// TwinCAT 3 PLC project P1
// ProgramVersion: 3.1.4024.0
// libraries:
//   Tc2_Standard, * (Beckhoff Automation GmbH)
//   Tc2_System, * (Beckhoff Automation GmbH)
//   Tc3_Module, * (Beckhoff Automation GmbH)
//   Tc3_PLCopen_OpcUa, * (Beckhoff Automation GmbH)
//   BeckhoffJsonReadWriter,1.0,fbarresi
// project tree:
//   Data_Types/ E_Errors2_ReactorSet.TcDUT, E_Errors_Module.TcDUT, E_Errors1_ReactorSet.TcDUT, E_Errors_Reactor.TcDUT, E_MachineState.TcDUT, E_PIDMode.TcDUT, E_ValveMode.TcDUT, ST_SeqResult_FAT.TcDUT, ST_Seq_FAT.TcDUT, ST_SeqSteps_FAT.TcDUT, ST_StepConfig_FAT.TcDUT, ST_StepSts_FAT.TcDUT
//   GVLs/ FAT.TcGVL, Global_Constants.TcGVL, Global_Variables.TcGVL, Set_Points_Interlocks.TcGVL
//   / PlcTask.TcTTO
//   POUs/ FB_Reactor.TcPOU, FB_Reactor_Set.TcPOU, FB_Reactor_Set_Ext_FAT.TcPOU, MAIN.TcPOU, P_Module.TcPOU
//   POUs/Functions/ F_AnalogIn.TcPOU, F_Concat3.TcPOU (not stored), F_Concat4.TcPOU (not stored), F_Error.TcPOU, F_Error_Check.TcPOU, F_Error_Range.TcPOU, F_IEConvert.TcPOU, F_LowestReal.TcPOU, F_HighestReal.TcPOU, F_Temperature.TcPOU
//   POUs/Function_Blocks/ FB_Door_Closed.TcPOU, FB_EdgeMonitor.TcPOU, FB_ReadWrite_Json.TcPOU, FB_ValveControl.TcPOU, FB_ValveStatus.TcPOU, FB_VFD.TcPOU, FB_Watchdog.TcPOU
// real-time tasks:
//   TASK PlcTask: cycle T#10ms, priority 20, ADS port 350
// I/O:
//   DEVICE Device 2 (EtherCAT Automation Protocol) (disabled), AmsNetId 10.0.2.15.2.1
//     Box 1 (Subscriber)
//     Box 2 (Publisher)
// variable links:
//   P1/P1 Instance <-> Device 2 (EtherCAT Automation Protocol)
//     PlcTask Inputs/P_Module.rs1.r1.fan_vfd_status <-> Inputs/DevState
//   P1/P1 Instance <-> Device 2 (EtherCAT Automation Protocol)/Box 1 (Subscriber)
//     PlcTask Inputs/P_Module.rs1.directive <-> RS1_Bytes/Inputs/VarData[0]
//     PlcTask Inputs/P_Module.rs1.rs_dead_air_pump_service_assigned <-> RS1_Bools/Inputs/VarData[1]
//     PlcTask Inputs/P_Module.rs1.rs_purge_assist_service_assigned <-> RS1_Bools/Inputs/VarData[3]
//     PlcTask Inputs/P_Module.rs1.rs_steam_system_service_assigned <-> RS1_Bools/Inputs/VarData[2]
//     PlcTask Inputs/P_Module.rs1.rs_vac_cooling_pump_service_assigned <-> RS1_Bools/Inputs/VarData[0]
//     PlcTask Inputs/P_Module.u_dead_air_pump_status <-> Module_Bytes/Inputs/VarData[1]
//     PlcTask Inputs/P_Module.u_module_generic_byte <-> Module_Bytes/Inputs/VarData[4]
//     PlcTask Inputs/P_Module.u_purge_assist_status <-> Module_Bytes/Inputs/VarData[3]
//     PlcTask Inputs/P_Module.u_steam_system_status <-> Module_Bytes/Inputs/VarData[2]
//     PlcTask Inputs/P_Module.u_vac_cooling_pump_status <-> Module_Bytes/Inputs/VarData[0]
//   P1/P1 Instance <-> Device 2 (EtherCAT Automation Protocol)/Box 2 (Publisher)
//     PlcTask Outputs/P_Module.rs1.r{1..4}.error_code <-> RS1_Dwords/Outputs/VarData[{1..4}]  (4 links)
//     PlcTask Outputs/P_Module.rs1.rs_adsorption <-> RS1_Bytes/Outputs/VarData[2]
//     PlcTask Outputs/P_Module.rs1.rs_air_repres <-> RS1_Bytes/Outputs/VarData[1]
//     PlcTask Outputs/P_Module.rs1.rs_dead_air_evac <-> RS1_Bytes/Outputs/VarData[3]
//     PlcTask Outputs/P_Module.rs1.rs_dead_air_pump_service_request <-> RS1_Bools/Outputs/VarData[1]
//     PlcTask Outputs/P_Module.rs1.rs_estop <-> RS1_Bytes/Outputs/VarData[6]
//     PlcTask Outputs/P_Module.rs1.rs_idle <-> RS1_Bytes/Outputs/VarData[0]
//     PlcTask Outputs/P_Module.rs1.rs_purge_assist_service_request <-> RS1_Bools/Outputs/VarData[3]
//     PlcTask Outputs/P_Module.rs1.rs_shutdown <-> RS1_Bytes/Outputs/VarData[7]
//     PlcTask Outputs/P_Module.rs1.rs_shutdown_evac <-> RS1_Bytes/Outputs/VarData[8]
//     PlcTask Outputs/P_Module.rs1.rs_steam_desorption <-> RS1_Bytes/Outputs/VarData[4]
//     PlcTask Outputs/P_Module.rs1.rs_steam_system_service_request <-> RS1_Bools/Outputs/VarData[2]
//     PlcTask Outputs/P_Module.rs1.rs_vac_cooling_pump_service_request <-> RS1_Bools/Outputs/VarData[0]
//     PlcTask Outputs/P_Module.rs1.rs_vacuum_cooling <-> RS1_Bytes/Outputs/VarData[5]

CONFIGURATION P1
    RESOURCE PLC ON TwinCAT3
        TASK PlcTask(INTERVAL := T#10ms, PRIORITY := 20);
        PROGRAM MAIN WITH PlcTask : MAIN;
    END_RESOURCE
END_CONFIGURATION

// ---- Data_Types/E_Errors2_ReactorSet.TcDUT
// P1 - E_Errors2_ReactorSet
// Rev 1.0 - October 31, 2024

TYPE E_Errors2_ReactorSet :
(
	errTBD								:= 0
);
END_TYPE

// ---- Data_Types/E_Errors_Module.TcDUT
// P1 - E_Errors_Module
// Rev 1.0 - October 15, 2024

TYPE E_Errors_Module :
(
	errInletCO2				         		:= 0,    
	errInletH2O,  
	errOutletH2O,			                 
	errSteamManifoldLinePres,    
	errFilterDiffPres,       
	errSorbentDiffPres,
	errReactorWallTemp,
	errInletAirTemp,
	errSteamTempNearRS1Temp,
	errSteamBypassValveNotInPos
);
END_TYPE

// ---- Data_Types/E_Errors1_ReactorSet.TcDUT
// P1 - E_Errors1_ReactorSet
// Rev 1.0 - October 31, 2024

TYPE E_Errors1_ReactorSet :
(
	errReactor								:= 0,			       
	errFanDiffPres,			       
	errOutletCO2,		         
	errReactorSetPres,		    
	errDoorsClosed,	       
	errRepresValvePosition,	 
	errDeadAirValvePosition,	 
	errPurgeValvePosition,	 
	errCoolingValvePosition,	 
	errSteamControlValvePosition,	 
	errSteamHeaderValvePosition,	 
	errDeadAirPumpServiceAssignmentLost,
	errPurgeAssistServiceAssignmentLost,
	errVacCoolingPumpServiceAssignmentLost,
	errSteamSystemServiceAssignmentLost,
	errAdsorptionFailedToCool,
	errEvacuationPresFailedToReachTarget,
	errReactorAboveMaxStoragePres,
	errReactorAboveMaxPres,
	errSorbentAboveMaxStorageTemp,
	errSorbentAboveMaxTemp,
	errInletTempAboveMaxAllowedTemp,	
	errInletTempBelowMinAllowedTemp,
	errInsufficientDesorptionVacuum,
	errInsufficientReactorPressure,
	errSteamRepressurizationOverPressure,
	errCoolingPressureTooHigh,
	errDeadAirValveSorbentTempTooHigh,
	errRepresValveSorbentTempTooHigh,
	errSteamHeaderValvePressureTooHigh,
	errRepresValveSteamValveOpen,
	errReactorLeak
);
END_TYPE

// ---- Data_Types/E_Errors_Reactor.TcDUT
// P1 - E_Errors_Reactor
// Rev 1.0 - October 15, 2024

TYPE E_Errors_Reactor :
(
	errInletDoorsClose						:= 0,
	errOutletDoorsClose,	
	errInletDoorsOpen,
	errOutletDoorsOpen,	
	errInletClampsRetract,	
	errOutletClampsRetract,
	errInletClampsExtend,
	errOutletClampsExtend,	
	errOutletLineTemp,
	errInletTopLeftTemp,		
	errInletTopRightTemp,	
	errInletBottomLeftTemp,	
	errInletBottomRightTemp,	
	errOutletTopLeftTemp,
	errOutletTopRightTemp,	
	errOutletBottomLeftTemp,	
	errOutletBottomRightTemp,
	errInletDoorsNotClosedForClamps,
	errOutletDoorsNotClosedForClamps,
	errInletClampsNotRetractedForDoors,
	errOutletClampsNotRetractedForDoors,
	errFanVFD,
	errFanRun
);
END_TYPE

// ---- Data_Types/E_MachineState.TcDUT
// P1 - E_MachineState
// Rev 1.0 - October 9, 2024

TYPE E_MachineState :
(
	eIdle						:= 0,
	eDeadAirEvacuation,
	eSteamDesorption,
	eVacuumCooling,
	eAirRepressurization,
	eAdsorption,
	eShutdown					:= 12,
	eShutdownEvac,
	eEmergencyStop
);
END_TYPE

// ---- Data_Types/E_PIDMode.TcDUT
// E_PIDMode
// Rev 1.0 - October 23, 2024

TYPE E_PIDMode :
(
	eOff						:= 0,
	eManual,
	eAuto,
	eTune
);
END_TYPE

// ---- Data_Types/E_ValveMode.TcDUT
// E_ValveMode
// Rev 1.0 - October 15, 2024

TYPE E_ValveMode :
(
	eClear						:= 0,
	eTransit,
	eError
);
END_TYPE

// ---- Data_Types/ST_SeqResult_FAT.TcDUT
TYPE ST_SeqResult_FAT :
STRUCT
	{attribute 'json' := 'TestName'}
	test_name : STRING;
	{attribute 'json' := 'TestDate'}
	test_date : STRING;
	{attribute 'json' := 'SeqSts'}
	status : STRING;
	{attribute 'json' := 'StepsCompleted'}
	steps : STRING;
	{attribute 'json' := 'error_id'}
	error : INT;
END_STRUCT
END_TYPE

// ---- Data_Types/ST_Seq_FAT.TcDUT
TYPE ST_Seq_FAT :
STRUCT
	{attribute 'json' := 'TestName'}
	test_name : STRING;
	{attribute 'json' := 'Step1'}
	step_1 : ST_SeqSteps_FAT;
	{attribute 'json' := 'Step2'}
	step_2 : ST_SeqSteps_FAT;
	{attribute 'json' := 'Step3'}
	step_3 : ST_SeqSteps_FAT;
	{attribute 'json' := 'Step4'}
	step_4 : ST_SeqSteps_FAT;
	{attribute 'json' := 'Step5'}
	step_5 : ST_SeqSteps_FAT;
	{attribute 'json' := 'Step6'}
	step_6 : ST_SeqSteps_FAT;
	{attribute 'json' := 'Step7'}
	step_7 : ST_SeqSteps_FAT;
	{attribute 'json' := 'Step8'}
	step_8 : ST_SeqSteps_FAT;
	{attribute 'json' := 'Step9'}
	step_9 : ST_SeqSteps_FAT;
	{attribute 'json' := 'Step10'}
	step_10 : ST_SeqSteps_FAT;
	
	
	
END_STRUCT
END_TYPE

// ---- Data_Types/ST_SeqSteps_FAT.TcDUT
TYPE ST_SeqSteps_FAT :
STRUCT
	{attribute 'json' := 'Summary'}
	summary : STRING(255);
	{attribute 'json' := 'Config'}
	config : ST_StepConfig_FAT;
END_STRUCT
END_TYPE

// ---- Data_Types/ST_StepConfig_FAT.TcDUT
TYPE ST_StepConfig_FAT :
STRUCT
	{attribute 'json' := 'react_pres'}
	react_press : REAL;
	{attribute 'json' := 'sorbent_temp'}
	sorbent_temp : REAL;
	{attribute 'json' := 'SP_1'}
	sp_1 : REAL;
	{attribute 'json' := 'SP_2'}
	sp_2 : REAL;
	{attribute 'json' := 'SP_3'}
	sp_3 : REAL;
	{attribute 'json' := 'SP_4'}
	sp_4 : REAL;
	{attribute 'json' := 'V_1'}
	valve_1 : STRING;
	{attribute 'json' := 'V_2'}
	valve_2 : STRING;
	{attribute 'json' := 'V_3'}
	valve_3 : STRING;
	{attribute 'json' := 'V_4'}
	valve_4 : STRING;
	{attribute 'json' := 'C_1'}
	check_1 : STRING;
	{attribute 'json' := 'C_2'}
	check_2 : STRING;
	{attribute 'json' := 'C_3'}
	check_3 : STRING;
	{attribute 'json' := 'C_4'}
	check_4 : STRING;
END_STRUCT
END_TYPE

// ---- Data_Types/ST_StepSts_FAT.TcDUT
TYPE ST_StepSts_FAT :
STRUCT
	{attribute 'json' := 'step_number'}
	step_number : INT;
	{attribute 'json' := 'react_pres'}
	react_press : REAL;
	{attribute 'json' := 'sorbent_temp'}
	sorbent_temp : REAL;
	{attribute 'json' := 'seq_sts'}
	seq_sts : STRING;
	
END_STRUCT
END_TYPE

// ---- GVLs/FAT.TcGVL
{attribute 'qualified_only'}
VAR_GLOBAL
	st_steam_desorption : ST_Seq_FAT;  // structure that parses the json file
	st_steam_desorption_result : ST_SeqResult_FAT;
	json_file_path : STRING(255) := 'C:/Users/asita/Documents/Steam_Desorption_FAT_Nominal.json';
END_VAR

// ---- GVLs/Global_Constants.TcGVL
// P1 - Global_Constants
// Rev 1.0 - November 2, 2024

VAR_GLOBAL CONSTANT
	
	_IDLE																: BYTE		:= 0;
	_STARTED															: BYTE		:= 1;
	_COMPLETED															: BYTE		:= 2;
	_ERROR																: BYTE		:= 9;
	
	_OPEN																: INT 		:= 100;
	_CLOSE																: INT		:= 0;
	
	_TEMP_VALID_TIME													: INT		:= 30;
	_VALVE_CHECK_TIME													: INT		:= 3000;

	_SECONDS															: REAL		:= 1000;
	_MINUTES															: REAL		:= 60000;
	
	_PERCENT_FACTOR														: REAL		:= 327.67;		// Factor to convert input to output percentage
	_VALVE_CLOSED														: INT		:= 3;
	_VALVE_OPEN															: INT		:= 95;

	_FAN_SPEED_MAX														: REAL		:= 1765;		// Maximum Fan RPM
	_FAN_SPEED_MIN														: REAL		:= 300;			// Minimum Fan RPM
	_FAN_ON																: REAL		:= 100;
	_FAN_START_TIME														: TIME		:= T#10S; 
	
	_DOOR_LATCH_CLOSE_TIME												: TIME		:= T#2S;

	_FAN_DELAY_TIME														: INT		:= 2000;
	_STOPPING_TIME														: REAL		:= 2000;

(*
	_DRAIN_TIME															: TIME		:= T#3S;
	_PUMP_SPEED_MAX														: REAL		:= 3540;		// Maximum Pump RPM
	_PUMP_SPEED_MIN														: REAL		:= 200;			// Minimum Pump RPM
	_FAN_RS_DELAY_TIME													: INT		:= 10000;
	_PAUSE_TIME															: REAL		:= 2000;
	_VALVE_TIME															: REAL		:= 3000;
	_FAN_SHUTDOWN_TIME													: REAL		:= 10000;
	_VALVE_INCREMENT_TIME												: REAL		:= 250;			// Time period for incremental change in valve position (mSecs)
	_VALVE_CLOSED														: INT		:= 3;
	_VALVE_OPEN															: INT		:= 95;
*)	
	_CURRENT_480_FACTOR													: REAL		:= 218.44;      // = 32767 counts / 150 amps
	_VOLTAGE_480_FACTOR													: REAL		:= 65.53;		// 0 - 500 VAC 
	_FAN_RPM_FACTOR														: REAL		:= 17.65;		// Factor to convert fan percent input to rpm output (max rpm / 100)

END_VAR

// ---- GVLs/Global_Variables.TcGVL
// P1 - Global_Variables
// Rev 1.0 - October 23, 2024

VAR_GLOBAL
	grDoorDelay															: REAL;
	grValveDelay														: REAL;
	grSteamControlValveDelay											: REAL;
	grClampDelay														: REAL;
	
	gbReset																: BOOL;
END_VAR

// ---- GVLs/Set_Points_Interlocks.TcGVL
// P1 - Set_Points_Interlocks
// Rev 1.0 - October 31, 2024

VAR_GLOBAL PERSISTENT
	
	{attribute 'OPC.UA.DA' := '1'}
	{attribute 'OPC.UA.DA.Access' := '1'}  				                
	IL_repres_valve_steam_valve_or										: BOOL;
	
	{attribute 'OPC.UA.DA' := '1'}
	SP_acceptable_reactor_pressure										: REAL;
	{attribute 'OPC.UA.DA' := '1'}
	SP_cooling_acceptable_pressure										: REAL;	
	{attribute 'OPC.UA.DA' := '1'}
	SP_cooling_target_pressure											: REAL;	
	{attribute 'OPC.UA.DA' := '1'}
	SP_clamp_extend_retract_duration									: REAL		:= 6;	
	{attribute 'OPC.UA.DA' := '1'}
	SP_door_open_close_duration											: REAL		:= 30;
	{attribute 'OPC.UA.DA' := '1'}
	SP_door_close_retries_before_error									: INT		:= 3;
	{attribute 'OPC.UA.DA' := '1'}
	SP_door_close_reset_duration										: REAL		:= 5;
	{attribute 'OPC.UA.DA' := '1'}	
	SP_evacuation_leak_test_acceptable_leak								: REAL		:= 0.2;
	{attribute 'OPC.UA.DA' := '1'}	
	SP_evacuation_leak_test_active										: BOOL;
	{attribute 'OPC.UA.DA' := '1'}	
	SP_evacuation_leak_test_duration									: REAL		:= 60;
	{attribute 'OPC.UA.DA' := '1'}
	SP_evacuation_target_pressure										: REAL;
	{attribute 'OPC.UA.DA' := '1'}
	SP_maximum_cooling_duration											: REAL;			
	{attribute 'OPC.UA.DA' := '1'}
	SP_maximum_desorption_sorbent_temperature							: REAL;			
	{attribute 'OPC.UA.DA' := '1'}	
	SP_maximum_evac_storage_pressure									: REAL;
	{attribute 'OPC.UA.DA' := '1'}	
	SP_maximum_evac_storage_temperature									: REAL;
	{attribute 'OPC.UA.DA' := '1'}
	SP_maximum_evacuation_duration										: REAL;
	{attribute 'OPC.UA.DA' := '1'}
	SP_maximum_inlet_air_temperature_during_adsorption					: REAL;						
	{attribute 'OPC.UA.DA' := '1'}
	SP_maximum_inlet_air_temperature									: REAL;
	{attribute 'OPC.UA.DA' := '1'}
	SP_maximum_pressure_for_steam_introduction							: REAL;
	{attribute 'OPC.UA.DA' := '1'}
	IL_maximum_pressure_for_steam_introduction_or						: BOOL;
	{attribute 'OPC.UA.DA' := '1'}
	{attribute 'OPC.UA.DA.Access' := '1'}  				                
	IL_maximum_pressure_for_steam_introduction_or_status				: BOOL;
	{attribute 'OPC.UA.DA' := '1'}
	SP_maximum_reactor_pressure											: REAL		:= 1.07;
	{attribute 'OPC.UA.DA' := '1'}
	IL_maximum_reactor_pressure_or										: BOOL;
	{attribute 'OPC.UA.DA' := '1'}
	{attribute 'OPC.UA.DA.Access' := '1'}  				                
	IL_maximum_reactor_pressure_or_status								: BOOL;
	{attribute 'OPC.UA.DA' := '1'}
	SP_maximum_reasonable_sorbent_TC_reading							: REAL;
	{attribute 'OPC.UA.DA' := '1'}
	SP_maximum_sorbent_temperature										: REAL;
	{attribute 'OPC.UA.DA' := '1'}
	IL_maximum_sorbent_temperature_or									: BOOL;
	{attribute 'OPC.UA.DA' := '1'}
	{attribute 'OPC.UA.DA.Access' := '1'}  				                
	IL_maximum_sorbent_temperature_or_status							: BOOL;
	{attribute 'OPC.UA.DA' := '1'}
	SP_maximum_sorbent_temperature_for_dead_air_line					: REAL;
	{attribute 'OPC.UA.DA' := '1'}
	IL_maximum_sorbent_temperature_for_dead_air_line_or					: BOOL;
	{attribute 'OPC.UA.DA' := '1'}
	{attribute 'OPC.UA.DA.Access' := '1'}  				                
	IL_maximum_sorbent_temperature_for_dead_air_line_or_status			: BOOL;
	{attribute 'OPC.UA.DA' := '1'}
	SP_maximum_sorbent_temperature_for_repressurization					: REAL;
	{attribute 'OPC.UA.DA' := '1'}
	IL_maximum_sorbent_temperature_for_repressurization_or				: BOOL;
	{attribute 'OPC.UA.DA' := '1'}
	{attribute 'OPC.UA.DA.Access' := '1'}  				                
	IL_maximum_sorbent_temperature_for_repressurization_or_status		: BOOL;
	{attribute 'OPC.UA.DA' := '1'}
	SP_maximum_steam_repressurization_duration							: REAL;
	{attribute 'OPC.UA.DA' := '1'}
	SP_minimum_evacuation_duration										: REAL;
	{attribute 'OPC.UA.DA' := '1'}
	SP_minimum_inlet_air_temperature									: REAL;
	{attribute 'OPC.UA.DA' := '1'}
	SP_minimum_reasonable_sorbent_TC_reading							: REAL;
	{attribute 'OPC.UA.DA' := '1'}
	SP_purge_duration													: REAL;
	{attribute 'OPC.UA.DA' := '1'}
	SP_steam_control_valve_open_close_duration							: REAL		:= 20;
	{attribute 'OPC.UA.DA' := '1'}
	SP_steam_control_valve_slow_move_increment							: REAL		:= 0.5;
	{attribute 'OPC.UA.DA' := '1'}
	SP_steam_control_valve_slow_move_full_open							: REAL		:= 15;
	{attribute 'OPC.UA.DA' := '1'}
	SP_purge_target_pressure											: REAL;
	{attribute 'OPC.UA.DA' := '1'}
	SP_steam_repressurization_target_pressure							: REAL;
	{attribute 'OPC.UA.DA' := '1'}
	SP_sufficient_desorption_pressure									: REAL;
	{attribute 'OPC.UA.DA' := '1'}
	SP_vacuum_cooling_target_temperature								: REAL;
	{attribute 'OPC.UA.DA' := '1'}
	SP_valve_open_close_duration										: REAL		:= 4;

END_VAR

// ---- POUs/MAIN.TcPOU
PROGRAM MAIN
VAR
	{attribute 'OPC.UA.DA' := '1'}  				                
	{attribute 'OPC.UA.DA.Access' := '1'}  				                
	plc_version															: STRING;

	bHalfSecondPulse													: BOOL;
	tonHalfSecPulse														: TON;
END_VAR

// P1 - Main
// Rev 1.0 - October 11, 2024

plc_version																:= '24_10_21_01';

/// TIMER PULSE
IF tonHalfSecPulse.Q THEN
	bHalfSecondPulse													:= NOT bHalfSecondPulse;
	tonHalfSecPulse(IN:= FALSE);
END_IF
tonHalfSecPulse(IN:= TRUE, PT:= T#500MS);

P_Module();

END_PROGRAM

// ---- POUs/P_Module.TcPOU
PROGRAM P_Module
VAR_INPUT
	
    /// <summary>XV08</summary>
	{attribute 'OPC.UA.DA' := '1'}  				                
	steam_bypass_valve													: BOOL;

    /// <summary>AT01 pump</summary>
	{attribute 'OPC.UA.DA' := '1'}  				                
	inlet_co2_pump														: BOOL;
	
    /// <summary>AT01 solenoid</summary>
	{attribute 'OPC.UA.DA' := '1'}  				                
	inlet_co2_sol														: BOOL;
	
END_VAR
VAR_OUTPUT
	test			: BOOL;
	/// EAP Variables
	m_error_code												AT %Q*	: DWORD;
	
	u_vac_cooling_pump_status									AT %I*	: BYTE;
	u_dead_air_pump_status										AT %I*	: BYTE;
	u_steam_system_status										AT %I*	: BYTE;
	u_purge_assist_status										AT %I*	: BYTE;
	u_instrument_air_status										AT %I*	: BYTE;
	u_module_generic_byte										AT %I*	: BYTE;
	
    /// <summary>XV08</summary>
	{attribute 'OPC.UA.DA' := '1'}  				                
	{attribute 'OPC.UA.DA.Access' := '1'}  				                
	steam_bypass_valve_cmd_status										: BOOL;
    /// <summary>XV08</summary>
	{attribute 'OPC.UA.DA' := '1'}  				                
	{attribute 'OPC.UA.DA.Access' := '1'}  				                
	steam_bypass_valve_status											: INT;
    /// <summary>XV08</summary>
	{attribute 'OPC.UA.DA' := '1'}  				                
	{attribute 'OPC.UA.DA.Access' := '1'}  				                
	steam_bypass_valve_open										AT %I*	: BOOL;
    /// <summary>XV08</summary>
	{attribute 'OPC.UA.DA' := '1'}  				                
	{attribute 'OPC.UA.DA.Access' := '1'}  				                
	steam_bypass_valve_closed									AT %I*	: BOOL;
	
    /// <summary>AT01 pump</summary>
	{attribute 'OPC.UA.DA' := '1'}  				                
	{attribute 'OPC.UA.DA.Access' := '1'}  				                
	inlet_co2_pump_cmd_status											: BOOL;
	
    /// <summary>AT01 solenoid</summary>
	{attribute 'OPC.UA.DA' := '1'}  				                
	{attribute 'OPC.UA.DA.Access' := '1'}  				                
	inlet_co2_sol_cmd_status											: BOOL;

	/// <summary>AT01</summary>
	{attribute 'OPC.UA.DA' := '1'}
	{attribute 'OPC.UA.DA.Access' := '1'}  				                
	inlet_co2															: REAL;
    /// <summary>AT01</summary>
	inlet_co2_error														: BOOL;

    /// <summary>AT02</summary>
	{attribute 'OPC.UA.DA' := '1'}  				                
	{attribute 'OPC.UA.DA.Access' := '1'}  				                
	inlet_h2o															: REAL;
    /// <summary>AT02</summary>
	inlet_h2o_error														: BOOL;

	/// <summary>AT04</summary>
	{attribute 'OPC.UA.DA' := '1'}  				                
	{attribute 'OPC.UA.DA.Access' := '1'}  				                
	outlet_h2o															: REAL;
    /// <summary>AT04</summary>
	outlet_h2o_error													: BOOL;

    /// <summary>PT02</summary>
	{attribute 'OPC.UA.DA' := '1'}  				                
	{attribute 'OPC.UA.DA.Access' := '1'}  				                
	steam_manifold_line_pres											: REAL;						
    /// <summary>PT02</summary>
	steam_manifold_line_pres_error 										: BOOL;

    /// <summary>PDT01</summary>
	{attribute 'OPC.UA.DA' := '1'}  				                
	{attribute 'OPC.UA.DA.Access' := '1'}  				                
	filter_diff_pres													: REAL;
    /// <summary>PDT01</summary>
	filter_diff_pres_error												: BOOL;

    /// <summary>PDT02</summary>
	{attribute 'OPC.UA.DA' := '1'}  				                
	{attribute 'OPC.UA.DA.Access' := '1'}  				                
	sorbent_diff_pres													: REAL;
    /// <summary>PDT02</summary>
	
    /// <summary>TT05</summary>
	{attribute 'OPC.UA.DA' := '1'}  				                
	{attribute 'OPC.UA.DA.Access' := '1'}  				                
	reactor_wall_temp													: REAL;						
    /// <summary>TT05</summary>
	reactor_wall_temp_error												: BOOL;						

    /// <summary>TT10</summary>
	{attribute 'OPC.UA.DA' := '1'}  				                
	{attribute 'OPC.UA.DA.Access' := '1'}  				                
	steam_temp_near_rs1													: REAL;						
    /// <summary>TT10</summary>
	steam_temp_near_rs1_error 											: BOOL;

    /// <summary>TT11</summary>
	{attribute 'OPC.UA.DA' := '1'}  				                
	{attribute 'OPC.UA.DA.Access' := '1'}  				                
	inlet_air_temp														: REAL;						
    /// <summary>TT11</summary>
	inlet_air_temp_error												: BOOL;						

END_VAR
VAR

	rs1																	: FB_Reactor_Set();
	//rs1																	: FB_Reactor_Set_Ext_FAT();
	//rs2																	: FB_Reactor_Set();
	//rs3																	: FB_Reactor_Set();
	
	fb_ReadJsonFAT : FB_ReadWrite_Json;
	sita_bit1 : BOOL;
	
	fbSteamBypassValve													: FB_valveStatus();
	
	rtrigReset															: R_TRIG;

    /// <summary>steam_bypass_valve</summary>
	XV_08														AT %Q*	: BOOL;
	
    /// <summary>Inlet CO2 pump</summary>
	AT01_pump													AT %Q*	: BOOL;
	
    /// <summary>Inlet CO2 solenoid</summary>
	AT01_sol													AT %Q*	: BOOL;

    /// <summary>Inlet CO2</summary>
	AT01														AT %I*	: INT;
    /// <summary>Inlet CO2</summary>
	{attribute 'OPC.UA.DA' := '1'}  				                
	{attribute 'OPC.UA.DA.Access' := '1'}  				                
	AT01_error													AT %I*	: BOOL;
    /// <summary>AT01</summary>
	{attribute 'OPC.UA.DA' := '1'}  				                
	inlet_co2_error_or													: BOOL;

    /// <summary>Inlet H2O</summary>
	AT02														AT %I*	: INT;
    /// <summary>Inlet H2O</summary>
	{attribute 'OPC.UA.DA' := '1'}  				                
	{attribute 'OPC.UA.DA.Access' := '1'}  				                
	AT02_error													AT %I*	: BOOL;
    /// <summary>AT02</summary>
	{attribute 'OPC.UA.DA' := '1'}  				                
	inlet_h2o_error_or													: BOOL;

    /// <summary>Outlet H20</summary>
	AT04														AT %I*	: INT;
    /// <summary>Outlet H2O</summary>
	{attribute 'OPC.UA.DA' := '1'}  				                
	{attribute 'OPC.UA.DA.Access' := '1'}  				                
	AT04_error													AT %I*	: BOOL;
    /// <summary>AT04</summary>
	{attribute 'OPC.UA.DA' := '1'}  				                
	outlet_h2o_error_or													: BOOL;

    /// <summary>steam manifold line pres</summary>
	PT02														AT %I*	: INT;
    /// <summary>steam manifold line pres</summary>
	{attribute 'OPC.UA.DA' := '1'}  				                
	{attribute 'OPC.UA.DA.Access' := '1'}  				                
	PT02_error													AT %I*	: BOOL;
    /// <summary>PT02</summary>
	{attribute 'OPC.UA.DA' := '1'}  				                
 	steam_manifold_line_pres_error_or									: BOOL;
	
    /// <summary>filter diff pres</summary>
	PDT01														AT %I*	: INT;
    /// <summary>filter diff pres</summary>
	{attribute 'OPC.UA.DA' := '1'}  				                
	{attribute 'OPC.UA.DA.Access' := '1'}  				                
	PDT01_error													AT %I*	: BOOL;
    /// <summary>PDT01</summary>
	{attribute 'OPC.UA.DA' := '1'}  				                
	filter_diff_pres_error_or											: BOOL;

	sorbent_diff_pres_error												: BOOL;
    /// <summary>sorbent diff pres</summary>
	PDT02														AT %I*	: INT;
    /// <summary>sorbent diff pres</summary>
	{attribute 'OPC.UA.DA' := '1'}  				                
	{attribute 'OPC.UA.DA.Access' := '1'}  				                
	PDT02_error													AT %I*	: BOOL;
    /// <summary>PDT02</summary>
	{attribute 'OPC.UA.DA' := '1'}  				                
	sorbent_diff_pres_error_or											: BOOL;

    /// <summary>reactor_wall_temp</summary>
	TT05														AT %I*	: INT;
    /// <summary>reactor_wall_temp</summary>
	{attribute 'OPC.UA.DA' := '1'}  				                
	{attribute 'OPC.UA.DA.Access' := '1'}  				                
	TT05_error													AT %I*	: BOOL;
    /// <summary>TT05</summary>
	{attribute 'OPC.UA.DA' := '1'}  				                
	reactor_wall_temp_error_or											: BOOL;
	
    /// <summary>steam temp near rs1</summary>
	TT10														AT %I*	: INT;
    /// <summary>steam temp near rs1</summary>
	{attribute 'OPC.UA.DA' := '1'}  				                
	{attribute 'OPC.UA.DA.Access' := '1'}  				                
	TT10_error													AT %I*	: BOOL;
    /// <summary>TT10</summary>
	{attribute 'OPC.UA.DA' := '1'}  				                
	steam_temp_near_rs01_error_or										: BOOL;           						

    /// <summary>inlet_air_temp</summary>
	TT11														AT %I*	: INT;
    /// <summary>inlet_air_temp</summary>
	{attribute 'OPC.UA.DA' := '1'}  				                
	{attribute 'OPC.UA.DA.Access' := '1'}  				                
	TT11_error													AT %I*	: BOOL;
    /// <summary>TT11/summary>
	{attribute 'OPC.UA.DA' := '1'}  				                
	inlet_air_temp_error_or												: BOOL;

	{attribute 'OPC.UA.DA' := '1'}  				                
	l1_current															: REAL;
	{attribute 'OPC.UA.DA' := '1'}  				                
	l1_current_error											AT %I*	: BOOL;
	IT_01														AT %I*	: INT;
	{attribute 'OPC.UA.DA' := '1'}  				                
	l2_current															: REAL;
	{attribute 'OPC.UA.DA' := '1'}  				                
	l2_current_error											AT %I*	: BOOL;
	IT_02														AT %I*	: INT;
	{attribute 'OPC.UA.DA' := '1'}  				                
	l3_current															: REAL;
	{attribute 'OPC.UA.DA' := '1'}  				                
	l3_current_error											AT %I*	: BOOL;
	IT_03														AT %I*	: INT;
	
	{attribute 'OPC.UA.DA' := '1'}  				                
	l1_voltage															: REAL;
	{attribute 'OPC.UA.DA' := '1'}  				                
	l1_volatge_error											AT %I*	: BOOL;
	VT_01														AT %I*	: INT;
	{attribute 'OPC.UA.DA' := '1'}  				                
	l2_voltage															: REAL;
	{attribute 'OPC.UA.DA' := '1'}  				                
	l2_volatge_error											AT %I*	: BOOL;
	VT_02														AT %I*	: INT;
	{attribute 'OPC.UA.DA' := '1'}  				                
	l3_voltage															: REAL;
	{attribute 'OPC.UA.DA' := '1'}  				                
	l3_volatge_error											AT %I*	: BOOL;
	VT_03														AT %I*	: INT;

END_VAR
	
{attribute 'qualified_only'}
VAR PERSISTENT

    /// <summary>PDT01</summary>
	{attribute 'OPC.UA.DA' := '1'}  				                
	filter_diff_pres_low												: REAL		:= 0;
    /// <summary>PDT01</summary>
	{attribute 'OPC.UA.DA' := '1'}  				                
	filter_diff_pres_high												: REAL		:= 1.5;
    /// <summary>PDT01</summary>
	{attribute 'OPC.UA.DA' := '1'}  				                
	filter_diff_pres_min												: REAL		:= 0.02;
    /// <summary>PDT01</summary>
	{attribute 'OPC.UA.DA' := '1'}  				                
	filter_diff_pres_offset												: REAL		:= 0;

    /// <summary>PDT02</summary>
	{attribute 'OPC.UA.DA' := '1'}  				                
	sorbent_diff_pres_low												: REAL		:= 0;
    /// <summary>PDT02</summary>
	{attribute 'OPC.UA.DA' := '1'}  				                
	sorbent_diff_pres_high												: REAL		:= 1.5;
    /// <summary>PDT02</summary>
	{attribute 'OPC.UA.DA' := '1'}  				                
	sorbent_diff_pres_min												: REAL		:= 0.02;
    /// <summary>PDT02</summary>
	{attribute 'OPC.UA.DA' := '1'}  				                
	sorbent_diff_pres_offset											: REAL		:= 0;

    /// <summary>AT01</summary>
	{attribute 'OPC.UA.DA' := '1'}  				                
	inlet_co2_low														: REAL		:= 0;
    /// <summary>AT01</summary>
	{attribute 'OPC.UA.DA' := '1'}  				                
	inlet_co2_high														: REAL		:= 2000;
    /// <summary>AT01</summary>
	{attribute 'OPC.UA.DA' := '1'}  				                
	inlet_co2_min														: REAL		:= 5;
    /// <summary>AT01</summary>
	{attribute 'OPC.UA.DA' := '1'}  				                
	inlet_co2_offset													: REAL		:= 0;

    /// <summary>AT02</summary>
	{attribute 'OPC.UA.DA' := '1'}  				                
	inlet_h2o_low														: REAL		:= 0;	  
    /// <summary>AT02</summary>                                                        
	{attribute 'OPC.UA.DA' := '1'}  				                                   
	inlet_h2o_high														: REAL		:= 2000;
    /// <summary>AT02</summary>                                                        
	{attribute 'OPC.UA.DA' := '1'}  				                                   
	inlet_h2o_min														: REAL		:= 5;	  
    /// <summary>AT02</summary>                                                        
	{attribute 'OPC.UA.DA' := '1'}  				                                   
	inlet_h2o_offset													: REAL		:= 0;	  

    /// <summary>AT04</summary>
	{attribute 'OPC.UA.DA' := '1'}  				                
	outlet_h2o_low														: REAL		:= 0;	  
    /// <summary>AT04</summary>                                                        
	{attribute 'OPC.UA.DA' := '1'}  				                                   
	outlet_h2o_high														: REAL		:= 2000;
    /// <summary>AT04</summary>                                                        
	{attribute 'OPC.UA.DA' := '1'}  				                                   
	outlet_h2o_min														: REAL		:= 5;	  
    /// <summary>AT04</summary>                                                        
	{attribute 'OPC.UA.DA' := '1'}  				                                   
	outlet_h2o_offset													: REAL		:= 0;	  

    /// <summary>PT02</summary>
	{attribute 'OPC.UA.DA' := '1'}  				                
	steam_manifold_line_pres_low										: REAL		:= 0;
    /// <summary>PT02</summary>
	{attribute 'OPC.UA.DA' := '1'}  				                
	steam_manifold_line_pres_high										: REAL		:= 2;
    /// <summary>PT02</summary>
	{attribute 'OPC.UA.DA' := '1'}  				                
	steam_manifold_line_pres_min										: REAL		:= 0;
    /// <summary>PT02</summary>
	{attribute 'OPC.UA.DA' := '1'}  				                
	steam_manifold_line_pres_offset										: REAL		:= 0;

    /// <summary>TT05</summary>
	{attribute 'OPC.UA.DA' := '1'}  				                
	reactor_wall_temp_offset											: REAL		:= 0;
    /// <summary>TT10</summary>
	{attribute 'OPC.UA.DA' := '1'}  				                
	steam_temp_near_rs1_offset											: REAL		:= 0;
    /// <summary>TT11</summary>
	{attribute 'OPC.UA.DA' := '1'}  				                
	inlet_air_temp_offset												: REAL		:= 0;
	
END_VAR

// P1 - P_Module
// Rev 1.0 - October 22, 2024

m_error_code															:= 0;

grDoorDelay																:= SP_door_open_close_duration * _SECONDS;
grValveDelay															:= SP_valve_open_close_duration * _SECONDS;
grSteamControlValveDelay												:= SP_steam_control_valve_open_close_duration * _SECONDS;
grClampDelay															:= SP_clamp_extend_retract_duration * _SECONDS;

gbReset																	:= FALSE;
rtrigReset(CLK:= BYTE_TO_INT(u_module_generic_byte) MOD 2 = 1);
IF rtrigReset.Q THEN
	gbReset																:= TRUE;
END_IF

XV_08																	:= steam_bypass_valve;
steam_bypass_valve_cmd_status											:= XV_08;
fbSteamBypassValve(Input:= steam_bypass_valve, Open:= steam_bypass_valve_open, Closed:= steam_bypass_valve_closed, Status=> steam_bypass_valve_status);
m_error_code															:= F_Error(m_error_code, steam_bypass_valve_status = eError, errSteamBypassValveNotInPos);

AT01_pump																:= inlet_co2_pump;
inlet_co2_pump_cmd_status												:= AT01_pump;

AT01_sol																:= inlet_co2_sol;
inlet_co2_sol_cmd_status												:= AT01_sol;

inlet_co2																:= F_AnalogIn(AT01, inlet_co2_low, inlet_co2_high, inlet_co2_min, inlet_co2_offset);
inlet_co2_error															:= AT01_error AND NOT inlet_co2_error_or;
m_error_code															:= F_Error(m_error_code, inlet_co2_error, errInletCO2);

inlet_h2o																:= F_AnalogIn(AT02, inlet_h2o_low, inlet_h2o_high, inlet_h2o_min, inlet_h2o_offset);
inlet_h2o_error															:= AT02_error AND NOT inlet_h2o_error_or;
m_error_code															:= F_Error(m_error_code, inlet_h2o_error, errInletH2O);

outlet_h2o																:= F_AnalogIn(AT04, outlet_h2o_low, outlet_h2o_high, outlet_h2o_min, outlet_h2o_offset);
outlet_h2o_error														:= AT04_error AND NOT outlet_h2o_error_or;
m_error_code															:= F_Error(m_error_code, outlet_h2o_error, errOutletH2O);

steam_manifold_line_pres												:= F_AnalogIn(PT02, steam_manifold_line_pres_low, steam_manifold_line_pres_high, steam_manifold_line_pres_min, steam_manifold_line_pres_offset);
steam_manifold_line_pres_error											:= PT02_Error AND NOT steam_manifold_line_pres_error_or;
m_error_code															:= F_Error(m_error_code, steam_manifold_line_pres_error, errSteamManifoldLinePres);

filter_diff_pres														:= F_AnalogIn(PDT01, filter_diff_pres_low, filter_diff_pres_high, filter_diff_pres_min, filter_diff_pres_offset);
filter_diff_pres_error													:= PDT01_error AND NOT filter_diff_pres_error_or; 
m_error_code															:= F_Error(m_error_code, filter_diff_pres_error, errFilterDiffPres);

sorbent_diff_pres														:= F_AnalogIn(PDT02, sorbent_diff_pres_low, sorbent_diff_pres_high, sorbent_diff_pres_min, sorbent_diff_pres_offset);
sorbent_diff_pres_error													:= PDT02_error AND NOT sorbent_diff_pres_error_or; 
m_error_code															:= F_Error(m_error_code, sorbent_diff_pres_error, errSorbentDiffPres);

reactor_wall_temp														:= F_Temperature(TT05, reactor_wall_temp_offset);
reactor_wall_temp_error													:= TT05_error AND NOT reactor_wall_temp_error_or;
m_error_code															:= F_Error(m_error_code, reactor_wall_temp_error, errReactorWallTemp);

steam_temp_near_rs1														:= F_Temperature(TT10, steam_temp_near_rs1_offset);
steam_temp_near_rs1_error												:= TT10_error AND NOT steam_temp_near_rs01_error_or;
m_error_code															:= F_Error(m_error_code, steam_temp_near_rs1_error, errSteamTempNearRS1Temp);

inlet_air_temp															:= F_Temperature(TT11, inlet_air_temp_offset);
inlet_air_temp_error													:= TT11_error AND NOT inlet_air_temp_error_or;
m_error_code															:= F_Error(m_error_code, inlet_air_temp_error, errInletAirTemp);

// ignore if < 2 Amps
l1_current																:= SEL(IT_01 > _CURRENT_480_FACTOR * 2, 0, F_IEConvert(IT_01, _CURRENT_480_FACTOR));
l2_current																:= SEL(IT_02 > _CURRENT_480_FACTOR * 2, 0, F_IEConvert(IT_02, _CURRENT_480_FACTOR));
l3_current																:= SEL(IT_03 > _CURRENT_480_FACTOR * 2, 0, F_IEConvert(IT_03, _CURRENT_480_FACTOR));

l1_voltage																:= F_IEConvert(VT_01, _VOLTAGE_480_FACTOR);
l2_voltage																:= F_IEConvert(VT_02, _VOLTAGE_480_FACTOR);
l3_voltage																:= F_IEConvert(VT_03, _VOLTAGE_480_FACTOR);

rs1(reactor_set	:= 1);
//rs2(reactor_set	:= 2);
//rs3(reactor_set	:= 3);

FAT_ReadWrite_Json();

METHOD FAT_ReadWrite_Json : BOOL
VAR_INPUT
END_VAR
fb_ReadJsonFAT(
		i_ExecuteRead := sita_bit1,
		i_Json_FilePath := FAT.json_file_path,
		i_JsonStructure := 'FAT.st_steam_desorption');
END_METHOD

END_PROGRAM

// ---- POUs/FB_Reactor_Set.TcPOU
FUNCTION_BLOCK FB_Reactor_Set
VAR_INPUT
	reactor_set															: INT;
END_VAR
VAR_OUTPUT
	bReset																: BOOL;
END_VAR
VAR
	/// EAP Variables
	power_up															: BYTE :=1;
	
	directive													AT %I*	: BYTE;	
	
	rs_vac_cooling_pump_service_assigned						AT %I*	: BOOL;
	rs_dead_air_pump_service_assigned							AT %I*	: BOOL;
	rs_steam_system_service_assigned							AT %I*	: BOOL;
	rs_purge_assist_service_assigned							AT %I*	: BOOL;
	rs_error_reset												AT %I*	: BOOL;

	rs_vac_cooling_pump_service_request							AT %Q*	: BOOL;
	rs_dead_air_pump_service_request							AT %Q*	: BOOL;
	rs_steam_system_service_request								AT %Q*	: BOOL;
	rs_purge_assist_service_request								AT %Q*	: BOOL;

	rs_idle														AT %Q*	: BYTE;
	rs_air_repres												AT %Q*	: BYTE;
	rs_adsorption												AT %Q*	: BYTE;
	rs_dead_air_evac											AT %Q*	: BYTE;
	rs_steam_desorption											AT %Q*	: BYTE;
	rs_vacuum_cooling											AT %Q*	: BYTE;
	rs_shutdown													AT %Q*	: BYTE;
	rs_shutdown_evac											AT %Q*	: BYTE;
	rs_estop													AT %Q*	: BYTE;
	
	rs_error_step												AT %Q*	: DWORD;
	rs_error_code_1												AT %Q*	: DWORD;
	rs_error_code_2												AT %Q*	: DWORD;
	
	{attribute 'OPC.UA.DA' := '1'} 
	{attribute 'OPC.UA.DA.Access' := '1'}  				                
	eState																: E_MachineState;
	
	r1																	: FB_Reactor();
	r2																	: FB_Reactor();
	r3																	: FB_Reactor();
	r4																	: FB_Reactor();
	
	fbRepresValve														: FB_ValveStatus();
	fbDeadAirValve														: FB_ValveStatus();
	fbPurgeValve														: FB_ValveStatus();
	fbCoolingValve														: FB_ValveStatus();
	fbSteamHeaderValve													: FB_ValveStatus();
	fbSteamControlValve													: FB_ValveStatus();

	fbSteamControlValveOp												: FB_ValveControl();
	
	rtrigDirectiveChange												: R_TRIG;
	rtrigReset															: R_TRIG;

	tonTimer1															: TON;
	//tonTimer2															: TON;
	
	i																	: INT;
	iDirective															: INT;
	
	rFanSpeed															: REAL;
	rTime1																: REAL;
	rTime2																: REAL;
	rSorbentHighTemp													: REAL;
	rEvacLeakTestInitialPressure										: REAL;
	rSteamControlValveControlPoint										: REAL;
	rSteamControlValveSlowMoveIncrement									: REAL		:= 0.5;
	rSteamControlValveSlowMoveFullOpen									: REAL		:= 15;

	bSteamControlValveControlPointError									: BOOL;	
	bError																: BOOL;
	bTimer1																: BOOL;
	bResetFanSpeed														: BOOL;
	bFanError															: BOOL;
	bFansRunning														: BOOL;
	bVacCoolingPumpServiceAssigned										: BOOL;
	bDeadAirPumpServiceAssigned											: BOOL;
	bSteamSystemServiceAssigned											: BOOL;
	bPurgeAssistServiceAssigned											: BOOL;
	bCoolingFailedFirstTry												: BOOL;
	
	bILDeadAirValveSorbentTempOK										: BOOL;
	bILSteamHeaderValvePresOK											: BOOL;
	bILRepresValveSorbentTempOK											: BOOL;
	bILReactorPresOK													: BOOL;
	bILSorbentTempOK													: BOOL;
	bILRepresValveSteamValveOK											: BOOL;
	
	bCloseAllValves														: BOOL;
	bAllValvesClear														: BOOL;
	bValveError															: BOOL;
	
	bOpenAllDoors														: BOOL;
	bCloseAllDoors														: BOOL;
	bAllDoorsOpen														: BOOL;
	bAllDoorsClosed														: BOOL;
	
	bExtendAllClamps													: BOOL;
	bRetractAllClamps													: BOOL;
	bAllClampsExtended													: BOOL;
	bAllClampsRetracted													: BOOL;
	
	bAllDoorsOpenError													: BOOL;
	bAllDoorsCloseError													: BOOL;
	bAllClampsRetractError												: BOOL;
	bAllClampsExtendError												: BOOL;
	
	bPriorDirective														: BYTE;
	
    /// <summary>PDT03</summary>
	{attribute 'OPC.UA.DA' := '1'}  				                
	{attribute 'OPC.UA.DA.Access' := '1'}  				                
	fan_diff_pres														: REAL;
    /// <summary>PDT03</summary>
	fan_diff_pres_error													: BOOL;
    /// <summary>fan diff pres</summary>
	PDT03														AT %I*	: INT;
    /// <summary>fanter diff pres</summary>
	{attribute 'OPC.UA.DA' := '1'}  				                
	{attribute 'OPC.UA.DA.Access' := '1'}  				                
	PDT03_error													AT %I*	: BOOL;
    /// <summary>PDT03</summary>
	{attribute 'OPC.UA.DA' := '1'}  				                
	fan_diff_pres_error_or												: BOOL;
	
    /// <summary>PDT03</summary>
	{attribute 'OPC.UA.DA' := '1'}  				                
	fan_diff_pres_off											AT %Q*	: BOOL;
	rtrigPDT03Off														: R_TRIG;
    /// <summary>R1_PDT03</summary>
	{attribute 'OPC.UA.DA' := '1'}  				                
	fan_diff_pres_sv01											AT %Q*	: BOOL;
	rtrigPDT03SV01														: R_TRIG;
    /// <summary>R2_PDT03</summary>
	{attribute 'OPC.UA.DA' := '1'}  				                
	fan_diff_pres_sv02											AT %Q*	: BOOL;
	rtrigPDT03SV02														: R_TRIG;
    /// <summary>R3_PDT03</summary>
	{attribute 'OPC.UA.DA' := '1'}  				                
	fan_diff_pres_sv03											AT %Q*	: BOOL;
	rtrigPDT03SV03														: R_TRIG;
    /// <summary>R4_PDT03</summary>
	{attribute 'OPC.UA.DA' := '1'}  				                
	fan_diff_pres_sv04											AT %Q*	: BOOL;
	rtrigPDT03SV04														: R_TRIG;

	/// <summary>PT01</summary>
	{attribute 'OPC.UA.DA' := '1'}
	{attribute 'OPC.UA.DA.Access' := '1'}  				                
	reactor_pres														: REAL;
    /// <summary>PT01</summary>
	reactor_pres_error													: BOOL;
    /// <summary>Reactor Pressure</summary>
	PT01														AT %I*	: INT;
    /// <summary>Reactor Pressure</summary>
	{attribute 'OPC.UA.DA' := '1'}  				                
	{attribute 'OPC.UA.DA.Access' := '1'}  				                
	PT01_error													AT %I*	: BOOL;
    /// <summary>PT01</summary>
	{attribute 'OPC.UA.DA' := '1'}  				                
	reactor_pres_error_or												: BOOL;

    /// <summary>AT03</summary>
	{attribute 'OPC.UA.DA' := '1'}  				                
	{attribute 'OPC.UA.DA.Access' := '1'}  				                
	outlet_co2															: REAL;
    /// <summary>AT03</summary>
	outlet_co2_error													: BOOL;
    /// <summary>Outlet CO2</summary>
	AT03														AT %I*	: INT;
    /// <summary>Outlet CO2</summary>
	{attribute 'OPC.UA.DA' := '1'}  				                
	{attribute 'OPC.UA.DA.Access' := '1'}  				                
	AT03_Error													AT %I*	: BOOL;
    /// <summary>AT03</summary>
	{attribute 'OPC.UA.DA' := '1'}  				                
	outlet_co2_error_or													: BOOL;
	
     /// <summary>AT03</summary>
	{attribute 'OPC.UA.DA' := '1'}  				                
	outlet_co2_off												AT %Q*	: BOOL;
	rtrigAT03Off														: R_TRIG;
    /// <summary>R1_AT03</summary>
	{attribute 'OPC.UA.DA' := '1'}  				                
	outlet_co2_sv01												AT %Q*	: BOOL;
	rtrigAT03SV01														: R_TRIG;
    /// <summary>R2_AT03</summary>
	{attribute 'OPC.UA.DA' := '1'}  				                
	outlet_co2_sv02												AT %Q*	: BOOL;
	rtrigAT03SV02														: R_TRIG;
    /// <summary>R3_AT03</summary>
	{attribute 'OPC.UA.DA' := '1'}  				                
	outlet_co2_sv03												AT %Q*	: BOOL;
	rtrigAT03SV03														: R_TRIG;
    /// <summary>R4_AT03</summary>
	{attribute 'OPC.UA.DA' := '1'}  				                
	outlet_co2_sv04												AT %Q*	: BOOL;
	rtrigAT03SV04														: R_TRIG;

   /// <summary>AI04</summary>
	{attribute 'OPC.UA.DA' := '1'}  				                
	{attribute 'OPC.UA.DA.Access' := '1'}  				                
	outlet_h2o															: REAL;
    /// <summary>AI04</summary>
	outlet_h2o_error													: BOOL;
    /// <summary>Outlet H20</summary>
	AT04														AT %I*	: INT;
    /// <summary>Outlet H2O</summary>
	{attribute 'OPC.UA.DA' := '1'}  				                
	{attribute 'OPC.UA.DA.Access' := '1'}  				                
	AT04_error													AT %I*	: BOOL;
    /// <summary>AT01</summary>
	{attribute 'OPC.UA.DA' := '1'}  				                
	outlet_h2o_error_or													: BOOL;

	{attribute 'OPC.UA.DA' := '1'}  				                
	{attribute 'OPC.UA.DA.Access' := '1'}  				                
	remaining_time														: REAL;
	{attribute 'OPC.UA.DA' := '1'}  				                
	{attribute 'OPC.UA.DA.Access' := '1'}  				                
	current_step														: INT;

    /// <summary>AT03 pump</summary>
	{attribute 'OPC.UA.DA' := '1'}  				                
	outlet_co2_pump														: BOOL;
    /// <summary>AT03 pump</summary>
	{attribute 'OPC.UA.DA' := '1'}  				                
	{attribute 'OPC.UA.DA.Access' := '1'}  				                
	outlet_co2_pump_cmd_status											: BOOL;
    /// <summary>Inlet CO2 pump</summary>
	AT03_pump													AT %Q*	: BOOL;
    /// <summary>AT03 solenoid</summary>
	{attribute 'OPC.UA.DA' := '1'}  				                
	outlet_co2_sol														: BOOL;
    /// <summary>AT03 solenoid</summary>
	{attribute 'OPC.UA.DA' := '1'}  				                
	{attribute 'OPC.UA.DA.Access' := '1'}  				                
	outlet_co2_sol_cmd_status											: BOOL;
    /// <summary>Outlet CO2 solenoid</summary>
	AT03_sol													AT %Q*	: BOOL;

	{attribute 'OPC.UA.DA' := '1'}  				                
	{attribute 'OPC.UA.DA.Access' := '1'}  				                
	ti_Total_Cycle_Count												: DINT; 
	{attribute 'OPC.UA.DA' := '1'}  				                
	{attribute 'OPC.UA.DA.Access' := '1'}  				                
	ti_Cycle_Count														: INT; 
	{attribute 'OPC.UA.DA' := '1'}  				                
	{attribute 'OPC.UA.DA.Access' := '1'}  				                
	tr_Remaining_Time													: REAL;

    /// <summary>PWR-01</summary>
	{attribute 'OPC.UA.DA' := '1'}  				                
	power_control														: BOOL;
    /// <summary>PWR-01</summary>
	{attribute 'OPC.UA.DA' := '1'}  				                
	{attribute 'OPC.UA.DA.Access' := '1'}  				                
	power_control_status												: BOOL;
    /// <summary>power_cmd</summary>
	PWR_01														AT %Q*	: BOOL;
	circuit_breaker_no_feedback									AT %I*	: BOOL;
	circuit_breaker_nc_feedback									AT %I*	: BOOL;
	
    /// <summary>PCV01</summary>
	{attribute 'OPC.UA.DA' := '1'}  				                
	steam_control_valve													: REAL;
    /// <summary>PCV01</summary>
	{attribute 'OPC.UA.DA' := '1'}  				                
	steam_control_valve_setpoint										: REAL;
    /// <summary>PCV01</summary>
	{attribute 'OPC.UA.DA' := '1'}  				                
	steam_control_valve_control_point_error								: BOOL;
    /// <summary>PCV01</summary>
	{attribute 'OPC.UA.DA' := '1'}  				                
	steam_control_valve_status											: INT;
    /// <summary>PCV01</summary>
	{attribute 'OPC.UA.DA' := '1'}  				                
	{attribute 'OPC.UA.DA.Access' := '1'}  				                
	steam_control_valve_position										: REAL;
    /// <summary>rs steam control valve</summary>
	PCV_01														AT %Q*	: INT;
    /// <summary>rs steam control valve</summary>
	PCV_01_position												AT %I*	: INT;
    /// <summary>PCV01</summary>
	{attribute 'OPC.UA.DA' := '1'}  				                
	{attribute 'OPC.UA.DA.Access' := '1'}  				                
	steam_control_valve_closed											: BOOL;
    /// <summary>PCV01</summary>
	{attribute 'OPC.UA.DA' := '1'}  				                
	{attribute 'OPC.UA.DA.Access' := '1'}  				                
	steam_control_valve_open											: BOOL;
    /// <summary>PCV01</summary>
	{attribute 'OPC.UA.DA' := '1'}  				                
	steam_control_valve_mode											: INT;			
    /// <summary>PCV01</summary>
	{attribute 'OPC.UA.DA' := '1'}  				                
	{attribute 'OPC.UA.DA.Access' := '1'}  				                
	steam_control_valve_current_mode									: INT;			
    /// <summary>PCV01</summary>
	steam_control_valve_kp												: REAL		:= 0.01; 
    /// <summary>PCV01</summary>
	steam_control_valve_ki												: REAL		:= 0.01;
    /// <summary>PCV01</summary>
	steam_control_valve_loop_time										: REAL		:= 2000;
    /// <summary>PCV01</summary>
	steam_control_valve_iband											: REAL		:= 6;
    /// <summary>PCV01</summary>
	steam_control_valve_base											: INT		:= 13110;
    /// <summary>PCV01</summary>
	steam_control_valve_base_adjust										: INT		:= 10;
		                                	        	
    /// <summary>XV02</summary>
	{attribute 'OPC.UA.DA' := '1'}  				                
	repres_valve														: BOOL;
    /// <summary>XV02</summary>
	{attribute 'OPC.UA.DA' := '1'}  				                
	{attribute 'OPC.UA.DA.Access' := '1'}  				                
	repres_valve_open_cmd_status										: BOOL;
    /// <summary>XV02</summary>
	{attribute 'OPC.UA.DA' := '1'}  				                
	{attribute 'OPC.UA.DA.Access' := '1'}  				                
	repres_valve_open											AT %I*	: BOOL;
    /// <summary>XV02</summary>
	{attribute 'OPC.UA.DA' := '1'}  				                
	{attribute 'OPC.UA.DA.Access' := '1'}  				                
	repres_valve_closed											AT %I*	: BOOL;
    /// <summary>repres valve</summary>
	XV_02														AT %Q*	: BOOL;
    /// <summary>XV02</summary>
	{attribute 'OPC.UA.DA' := '1'}  				                
	{attribute 'OPC.UA.DA.Access' := '1'}  				                
	repres_valve_status													: INT;
	
    /// <summary>XV04</summary>
	{attribute 'OPC.UA.DA' := '1'}  				                
	dead_air_valve														: BOOL;
    /// <summary>XV04</summary>
	{attribute 'OPC.UA.DA' := '1'}  				                
	{attribute 'OPC.UA.DA.Access' := '1'}  				                
	dead_air_valve_open_cmd_status										: BOOL;
    /// <summary>XV04</summary>
	{attribute 'OPC.UA.DA' := '1'}  				                
	{attribute 'OPC.UA.DA.Access' := '1'}  				                
	dead_air_valve_open											AT %I*	: BOOL;
    /// <summary>XV04</summary>
	{attribute 'OPC.UA.DA' := '1'}  				                
	{attribute 'OPC.UA.DA.Access' := '1'}  				                
	dead_air_valve_closed										AT %I*	: BOOL;
    /// <summary>dead air valve</summary>
	XV_04														AT %Q*	: BOOL;
    /// <summary>XV04</summary>
	{attribute 'OPC.UA.DA' := '1'}  				                
	{attribute 'OPC.UA.DA.Access' := '1'}  				                
	dead_air_valve_status												: INT;
	
    /// <summary>XV05</summary>
	{attribute 'OPC.UA.DA' := '1'}  				                
	purge_valve															: BOOL;
    /// <summary>XV05</summary>
	{attribute 'OPC.UA.DA' := '1'}  				                
	{attribute 'OPC.UA.DA.Access' := '1'}  				                
	purge_valve_open_cmd_status											: BOOL;
    /// <summary>XV05</summary>
	{attribute 'OPC.UA.DA' := '1'}  				                
	{attribute 'OPC.UA.DA.Access' := '1'}  				                
	purge_valve_open											AT %I*	: BOOL;
    /// <summary>XV05</summary>
	{attribute 'OPC.UA.DA' := '1'}  				                
	{attribute 'OPC.UA.DA.Access' := '1'}  				                
	purge_valve_closed											AT %I*	: BOOL;
    /// <summary>purge valve</summary>
	XV_05														AT %Q*	: BOOL;
    /// <summary>XV05</summary>
	{attribute 'OPC.UA.DA' := '1'}  				                
	{attribute 'OPC.UA.DA.Access' := '1'}  				                
	purge_valve_status													: INT;
	
    /// <summary>XV06</summary>
	{attribute 'OPC.UA.DA' := '1'}  				                
	cooling_valve														: BOOL;
    /// <summary>XV06</summary>
	{attribute 'OPC.UA.DA' := '1'}  				                
	{attribute 'OPC.UA.DA.Access' := '1'}  				                
	cooling_valve_open_cmd_status										: BOOL;
    /// <summary>XV06</summary>
	{attribute 'OPC.UA.DA' := '1'}  				                
	{attribute 'OPC.UA.DA.Access' := '1'}  				                
	cooling_valve_open											AT %I*	: BOOL;
    /// <summary>XV06</summary>
	{attribute 'OPC.UA.DA' := '1'}  				                
	{attribute 'OPC.UA.DA.Access' := '1'}  				                
	cooling_valve_closed										AT %I*	: BOOL;
    /// <summary>cooling valve</summary>
	XV_06														AT %Q*	: BOOL;
    /// <summary>XV06</summary>
	{attribute 'OPC.UA.DA' := '1'}  				                
	{attribute 'OPC.UA.DA.Access' := '1'}  				                
	cooling_valve_status												: INT;
	
    /// <summary>XV07</summary>
	{attribute 'OPC.UA.DA' := '1'}  				                
	steam_header_valve													: BOOL;
    /// <summary>XV07</summary>
	{attribute 'OPC.UA.DA' := '1'}  				                
	{attribute 'OPC.UA.DA.Access' := '1'}  				                
	steam_header_valve_open_cmd_status									: BOOL;
    /// <summary>XV07</summary>
	{attribute 'OPC.UA.DA' := '1'}  				                
	{attribute 'OPC.UA.DA.Access' := '1'}  				                
	steam_header_valve_open										AT %I*	: BOOL;
    /// <summary>XV07</summary>
	{attribute 'OPC.UA.DA' := '1'}  				                
	{attribute 'OPC.UA.DA.Access' := '1'}  				                
	steam_header_valve_closed									AT %I*	: BOOL;
    /// <summary>steam header valve</summary>
	XV_07														AT %Q*	: BOOL;
    /// <summary>XV07</summary>
	{attribute 'OPC.UA.DA' := '1'}  				                
	{attribute 'OPC.UA.DA.Access' := '1'}  				                
	steam_header_valve_status											: INT;

END_VAR

VAR PERSISTENT
	
    /// <summary>AT03</summary>
	{attribute 'OPC.UA.DA' := '1'}  				                
	outlet_co2_low														: REAL	:= 0;
    /// <summary>AT03</summary>
	{attribute 'OPC.UA.DA' := '1'}  				                
	outlet_co2_high														: REAL	:= 2000;
    /// <summary>AT03</summary>
	{attribute 'OPC.UA.DA' := '1'}  				                
	outlet_co2_min														: REAL	:= 5;
    /// <summary>AT03</summary>
	{attribute 'OPC.UA.DA' := '1'}  				                
	outlet_co2_offset													: REAL	:= 0;

    /// <summary>PT03</summary>
	{attribute 'OPC.UA.DA' := '1'}  				                
	reactor_set_pres_low												: REAL	:= 0;
    /// <summary>PT03</summary>
	{attribute 'OPC.UA.DA' := '1'}  				                
	reactor_set_pres_high												: REAL	:= 2000;
    /// <summary>PT03</summary>
	{attribute 'OPC.UA.DA' := '1'}  				                
	reactor_set_pres_min												: REAL	:= 5;
    /// <summary>PT03</summary>
	{attribute 'OPC.UA.DA' := '1'}  				                
	reactor_set_pres_offset												: REAL	:= 0;

    /// <summary>PDT03</summary>
	{attribute 'OPC.UA.DA' := '1'}  				                
	fan_diff_pres_low													: REAL	:= 0;
    /// <summary>PDT03</summary>
	{attribute 'OPC.UA.DA' := '1'}  				                
	fan_diff_pres_high													: REAL	:= 1.5;
    /// <summary>PDT03</summary>
	{attribute 'OPC.UA.DA' := '1'}  				                
	fan_diff_pres_min													: REAL	:= 0.02;
    /// <summary>PDT03</summary>
	{attribute 'OPC.UA.DA' := '1'}  				                
	fan_diff_pres_offset												: REAL	:= 0;

END_VAR

// P1 - FB_Reactor_Set
// Rev 1.0 - October 31, 2024

bReset																	:= FALSE;
rtrigReset(CLK:= rs_error_reset);
IF rtrigReset.Q THEN
	bReset																:= TRUE;
	A_EAP_Reset();
END_IF

r1(unit	:= 1, reset	:= bReset);
r2(unit	:= 2, reset	:= bReset);
r3(unit	:= 3, reset	:= bReset);
r4(unit := 4, reset	:= bReset);

rs_error_code_1															:= SEL(bReset, rs_error_code_1, 0);

A_IO_ReactorSet();

rtrigDirectiveChange(CLK:= directive <> bPriorDirective);
IF rtrigDirectiveChange.Q THEN
	A_Eap_Reset();
	iDirective															:= BYTE_TO_INT(directive);
	estate																:= iDirective;
	current_step														:= 1;
	bPriorDirective														:= directive;
END_IF

CASE eState OF
	
	eIdle:
		rs_idle															:= _STARTED;
		current_step													:= 0;
		
	eDeadAirEvacuation:
		A_Process_Dead_Air_Evacuation();

	eSteamDesorption:
	
	Steam_Desorption_FAT(i_Execute := TRUE);
	A_Process_Steam_Desorption();
		
	eVacuumCooling:
		A_Process_Vacuum_Cooling();
		
	eAirRepressurization:
		A_Process_Air_Repressurization();
		
	eAdsorption:
		A_Process_Adsorption_1();
		
	eShutdown:
		A_Shutdown();

	eShutdownEvac:
		A_Shutdown_Evac();

	eEmergencyStop:
		A_Shutdown_Estop_1();

END_CASE

remaining_time															:= 0;
IF eState > eIdle THEN
	IF bTimer1 THEN
		remaining_time													:= rTime1 - TIME_TO_REAL(tonTimer1.ET);
	//ELSIF bTimer2 THEN
		//remaining_time													:= rTime2 - TIME_TO_REAL(tonTimer2.ET);
	END_IF
END_IF

tonTimer1(IN:= bTimer1, PT:= REAL_TO_TIME(rTime1));
//tonTimer2(IN:= bTimer2, PT:= REAL_TO_TIME(rTime2));


// FAT Tests

ACTION A_EAP_Reset:
// P1 - FB_Reactor_Set.A_EAP_Reset
// Rev 1.0 - October 22, 2024

rs_idle																	:= _IDLE;
rs_air_repres															:= _IDLE;
rs_adsorption															:= _IDLE;
rs_dead_air_evac														:= _IDLE;
rs_steam_desorption														:= _IDLE;
rs_vacuum_cooling														:= _IDLE;
rs_shutdown																:= _IDLE;
rs_shutdown_evac														:= _IDLE;
rs_estop																:= _IDLE;

A_EAP_Services_Reset();
END_ACTION

ACTION A_EAP_Services_Check:
// P1 - FB_Reactor_Set.A_EAP_Services_Check
// Rev 1.0 - October 31, 2024

IF bPurgeAssistServiceAssigned AND NOT rs_purge_assist_service_assigned THEN
	rs_error_code_1														:= F_Error(rs_error_code_1, TRUE, errPurgeAssistServiceAssignmentLost);
	M_Step(98);
ELSIF bVacCoolingPumpServiceAssigned AND NOT rs_vac_cooling_pump_service_assigned THEN
	rs_error_code_1														:= F_Error(rs_error_code_1, TRUE, errVacCoolingPumpServiceAssignmentLost);
	M_Step(98);
ELSIF bSteamSystemServiceAssigned AND NOT rs_steam_system_service_assigned THEN
	rs_error_code_1														:= F_Error(rs_error_code_1, TRUE, errSteamSystemServiceAssignmentLost);
	M_Step(98);
END_IF
END_ACTION

ACTION A_EAP_Services_Reset:
// P1 - FB_Reactor_Set.A_EAP_Services_Reset
// Rev 1.0 - October 22, 2024

rs_vac_cooling_pump_service_request										:= FALSE;
rs_dead_air_pump_service_request										:= FALSE;
rs_steam_system_service_request											:= FALSE;
rs_purge_assist_service_request											:= FALSE;
bVacCoolingPumpServiceAssigned											:= FALSE;
bDeadAirPumpServiceAssigned												:= FALSE;
bSteamSystemServiceAssigned												:= FALSE;
bPurgeAssistServiceAssigned												:= FALSE;
END_ACTION

ACTION A_IO_ReactorSet:
// P1 - FB_Reactor_Set.A_IO_ReactorSet
// Rev 1.0 - October 31, 2024

IL_maximum_sorbent_temperature_for_repressurization_or_status			:= IL_maximum_sorbent_temperature_for_repressurization_or;
IL_maximum_sorbent_temperature_for_dead_air_line_or_status				:= IL_maximum_sorbent_temperature_for_dead_air_line_or;
IL_maximum_pressure_for_steam_introduction_or_status					:= IL_maximum_pressure_for_steam_introduction_or;
IL_maximum_reactor_pressure_or_status									:= IL_maximum_reactor_pressure_or;
IL_maximum_sorbent_temperature_or_status								:= IL_maximum_sorbent_temperature_or;

IF bReset THEN
	rs_error_code_1														:= F_Error(rs_error_code_1, FALSE, errDeadAirValveSorbentTempTooHigh);		// Interlock 3
	rs_error_code_1														:= F_Error(rs_error_code_1, FALSE, errSteamHeaderValvePressureTooHigh);		// Interlock 4
	rs_error_code_1														:= F_Error(rs_error_code_1, FALSE, errRepresValveSorbentTempTooHigh);		// Interlock 5
	rs_error_code_1														:= F_Error(rs_error_code_1, FALSE, errRepresValveSteamValveOpen);			// Interlock 9
END_IF

IF bResetFanSpeed THEN
	r1.fan_vfd															:= rFanSpeed;
	r2.fan_vfd															:= rFanSpeed;
	r3.fan_vfd															:= rFanSpeed;
	r4.fan_vfd															:= rFanSpeed;
	bResetFanSpeed														:= FALSE;	
END_IF

bFanError																:= r1.fan_run_error OR r1.fan_vfd_error OR r2.fan_run_error OR r2.fan_vfd_error OR r3.fan_run_error OR r3.fan_vfd_error OR r4.fan_run_error OR r4.fan_vfd_error;
bFansRunning															:= r1.fan_running AND r2.fan_running AND r3.fan_running AND r4.fan_running;

rtrigPDT03Off(CLK:= fan_diff_pres_off);
rtrigPDT03SV01(CLK:= fan_diff_pres_sv01);
rtrigPDT03SV02(CLK:= fan_diff_pres_sv02);
rtrigPDT03SV03(CLK:= fan_diff_pres_sv03);
rtrigPDT03SV04(CLK:= fan_diff_pres_sv04);
IF rtrigPDT03Off.Q THEN
	fan_diff_pres_sv01													:= FALSE;
	fan_diff_pres_sv02													:= FALSE;
	fan_diff_pres_sv03													:= FALSE;
	fan_diff_pres_sv04													:= FALSE;
	fan_diff_pres_off													:= FALSE;
ELSIF rtrigPDT03SV01.Q THEN
	fan_diff_pres_sv02													:= FALSE;
	fan_diff_pres_sv03													:= FALSE;
	fan_diff_pres_sv04													:= FALSE;
ELSIF rtrigPDT03SV02.Q THEN
	fan_diff_pres_sv01													:= FALSE;
	fan_diff_pres_sv03													:= FALSE;
	fan_diff_pres_sv04													:= FALSE;
ELSIF rtrigPDT03SV03.Q THEN
	fan_diff_pres_sv01													:= FALSE;
	fan_diff_pres_sv02													:= FALSE;
	fan_diff_pres_sv04													:= FALSE;
ELSIF rtrigPDT03SV04.Q THEN
	fan_diff_pres_sv01													:= FALSE;
	fan_diff_pres_sv02													:= FALSE;
	fan_diff_pres_sv03													:= FALSE;
END_IF

rtrigAT03Off(CLK:= outlet_co2_off);
rtrigAT03SV01(CLK:= outlet_co2_sv01);
rtrigAT03SV02(CLK:= outlet_co2_sv02);
rtrigAT03SV03(CLK:= outlet_co2_sv03);
rtrigAT03SV04(CLK:= outlet_co2_sv04);
IF rtrigAT03Off.Q THEN
	outlet_co2_sv01														:= FALSE;
	outlet_co2_sv02														:= FALSE;
	outlet_co2_sv03														:= FALSE;
	outlet_co2_sv04														:= FALSE;
	outlet_co2_off														:= FALSE;
ELSIF rtrigAT03SV01.Q THEN
	outlet_co2_sv02														:= FALSE;
	outlet_co2_sv03														:= FALSE;
	outlet_co2_sv04														:= FALSE;
ELSIF rtrigAT03SV02.Q THEN
	outlet_co2_sv01														:= FALSE;
	outlet_co2_sv03														:= FALSE;
	outlet_co2_sv04														:= FALSE;
ELSIF rtrigAT03SV03.Q THEN
	outlet_co2_sv01														:= FALSE;
	outlet_co2_sv02														:= FALSE;
	outlet_co2_sv04														:= FALSE;
ELSIF rtrigAT03SV04.Q THEN
	outlet_co2_sv01														:= FALSE;
	outlet_co2_sv02														:= FALSE;
	outlet_co2_sv03														:= FALSE;
END_IF

fan_diff_pres															:= F_AnalogIn(PDT03, fan_diff_pres_low, fan_diff_pres_high, fan_diff_pres_min, fan_diff_pres_offset);
fan_diff_pres_error														:= PDT03_error AND NOT fan_diff_pres_error_or;
rs_error_code_1															:= F_Error(rs_error_code_1, fan_diff_pres_error, errFanDiffPres);

outlet_co2																:= F_AnalogIn(AT03, outlet_co2_low, outlet_co2_high, outlet_co2_min, outlet_co2_offset);
outlet_co2_error														:= AT03_error AND NOT outlet_co2_error_or;
rs_error_code_1															:= F_Error(rs_error_code_1, outlet_co2_error, errOutletCO2);

reactor_pres															:= F_AnalogIn(PT01, reactor_set_pres_low, reactor_set_pres_high, reactor_set_pres_min, reactor_set_pres_offset);
reactor_pres_error														:= PT01_error AND NOT reactor_pres_error_or;
rs_error_code_1															:= F_Error(rs_error_code_1, reactor_pres_error, errReactorSetPres);

// Interlock 6
bILReactorPresOK														:= reactor_pres <= SP_maximum_reactor_pressure OR IL_maximum_reactor_pressure_or;
rs_error_code_1															:= F_Error(rs_error_code_1, NOT bILReactorPresOK, errReactorAboveMaxPres);

IF bCloseAllValves THEN
	repres_valve														:= FALSE;
	dead_air_valve														:= FALSE;
	purge_valve															:= FALSE;
	cooling_valve														:= FALSE;
	steam_header_valve													:= FALSE;
	bCloseAllValves														:= FALSE;
END_IF

XV_02																	:= repres_valve;
repres_valve_open_cmd_status											:= XV_02;
fbRepresValve(Input:= repres_valve, Open:= repres_valve_open, Closed:= repres_valve_closed, Delay:= grValveDelay, Status=> repres_valve_status);
rs_error_code_1															:= F_Error(rs_error_code_1, repres_valve_status = eError, errRepresValvePosition);
// Interlock 5
bILRepresValveSorbentTempOK												:= rSorbentHighTemp <= SP_maximum_sorbent_temperature_for_repressurization OR IL_maximum_sorbent_temperature_for_repressurization_or;
IF rSorbentHighTemp <= SP_maximum_sorbent_temperature_for_repressurization THEN
	rs_error_code_1														:= F_Error(rs_error_code_1, FALSE, errRepresValveSorbentTempTooHigh);
END_IF
// Interlock 9
bILRepresValveSteamValveOK												:= steam_header_valve_closed OR IL_repres_valve_steam_valve_or;
IF steam_header_valve_closed THEN
	rs_error_code_1														:= F_Error(rs_error_code_1, FALSE, errRepresValveSteamValveOpen);
END_IF


XV_04																	:= dead_air_valve;
dead_air_valve_open_cmd_status											:= XV_04;
fbDeadAirValve(Input:= dead_air_valve, Open:= dead_air_valve_open, Closed:= dead_air_valve_closed, Delay:= grValveDelay, Status=> dead_air_valve_status);
rs_error_code_1															:= F_Error(rs_error_code_1, dead_air_valve_status = eError, errDeadAirValvePosition);
// Interlock 3
bILDeadAirValveSorbentTempOK											:= rSorbentHighTemp <= SP_maximum_sorbent_temperature_for_dead_air_line OR IL_maximum_sorbent_temperature_for_dead_air_line_or;
IF rSorbentHighTemp <= SP_maximum_sorbent_temperature_for_dead_air_line THEN
	rs_error_code_1														:= F_Error(rs_error_code_1, FALSE, errDeadAirValveSorbentTempTooHigh);
END_IF

XV_05																	:= purge_valve;
purge_valve_open_cmd_status												:= XV_05;
fbPurgeValve(Input:= purge_valve, Open:= purge_valve_open, Closed:= purge_valve_closed, Delay:= grValveDelay, Status=> purge_valve_status);
rs_error_code_1															:= F_Error(rs_error_code_1, purge_valve_status = eError, errPurgeValvePosition);

XV_06																	:= cooling_valve;
cooling_valve_open_cmd_status											:= XV_06;
fbCoolingValve(Input:= cooling_valve, Open:= cooling_valve_open, Closed:= cooling_valve_closed, Delay:= grValveDelay, Status=> cooling_valve_status);
rs_error_code_1															:= F_Error(rs_error_code_1, cooling_valve_status = eError, errCoolingValvePosition);

XV_07																	:= steam_header_valve;
steam_header_valve_open_cmd_status										:= XV_07;
fbSteamHeaderValve(Input:= steam_header_valve, Open:= steam_header_valve_open, Closed:= steam_header_valve_closed, Delay:= grValveDelay, Status=> steam_header_valve_status);
rs_error_code_1															:= F_Error(rs_error_code_1, steam_header_valve_status = eError, errSteamHeaderValvePosition);
// Interlock 4
bILSteamHeaderValvePresOK												:= reactor_pres <= SP_maximum_pressure_for_steam_introduction OR IL_maximum_pressure_for_steam_introduction_or;
IF reactor_pres <= SP_maximum_pressure_for_steam_introduction THEN
	rs_error_code_1														:= F_Error(rs_error_code_1, FALSE, errSteamHeaderValvePressureTooHigh);
END_IF

steam_control_valve_position											:= INT_TO_REAL(PCV_01_position) / _PERCENT_FACTOR; 
steam_control_valve_closed												:= steam_control_valve_position <= _VALVE_CLOSED;
steam_control_valve_open												:= steam_control_valve_position >= _VALVE_OPEN;

fbSteamControlValveOp(	Setpoint										:= steam_control_valve_setpoint,							// Set point for modulation control
						Control											:= rSteamControlValveControlPoint,							// Input controlling valve modulation
						Error											:= bSteamControlValveControlPointError,						// Error of input controlling modulation
						Closed											:= steam_control_valve_closed,								// Used to open valve slowly in manual mode
						Reverse											:= FALSE,													// Controls modulation direction
						Kp												:= steam_control_valve_kp,           						// Modulation control values
						Ki												:= steam_control_valve_ki,           
						BaseAdjust										:= steam_control_valve_base_adjust,  
						LoopTime										:= steam_control_valve_loop_time,    
						IBand											:= steam_control_valve_iband,        
						Base											:= steam_control_valve_base,         
						Mode											:= steam_control_valve_mode,
						Input											:= steam_control_valve,										// Manual control input
						Input_Increment									:= rSteamControlValveSlowMoveIncrement,
						Full_Output_SP									:= rSteamControlValveSlowMoveFullOpen,
						Mode_Out										=> steam_control_valve_current_mode, 
						Output											=> PCV_01);

IF steam_control_valve_current_mode = eManual AND (steam_control_valve = _OPEN OR steam_control_valve = _CLOSE) THEN
	fbSteamControlValve(Input:= steam_control_valve = _OPEN, Open:= steam_control_valve_open, Closed:= steam_control_valve_closed, Delay:= grSteamControlValveDelay, Status=> steam_control_valve_status);
ELSE
	steam_control_valve_status											:= eClear;
END_IF
rs_error_code_1															:= F_Error(rs_error_code_1, steam_control_valve_status = eError, errSteamControlValvePosition);

bAllValvesClear															:= repres_valve_status + dead_air_valve_status + purge_valve_status + cooling_valve_status + steam_header_valve_status = eClear;
bValveError																:= repres_valve_status = eError OR dead_air_valve_status = eError OR purge_valve_status = eError OR cooling_valve_status = eError OR steam_header_valve_status = eError;

IF bOpenAllDoors THEN
	r1.open_inlet_doors													:= TRUE;
	r2.open_inlet_doors													:= TRUE;
	r3.open_inlet_doors													:= TRUE;
	r4.open_inlet_doors													:= TRUE;
	r1.open_outlet_doors												:= TRUE;
	r2.open_outlet_doors												:= TRUE;
	r3.open_outlet_doors												:= TRUE;
	r4.open_outlet_doors												:= TRUE;
	bOpenAllDoors														:= FALSE;
END_IF
	
IF bCloseAllDoors THEN
	r1.close_inlet_doors												:= TRUE;
	r2.close_inlet_doors												:= TRUE;
	r3.close_inlet_doors												:= TRUE;
	r4.close_inlet_doors												:= TRUE;
	r1.close_outlet_doors												:= TRUE;
	r2.close_outlet_doors												:= TRUE;
	r3.close_outlet_doors												:= TRUE;
	r4.close_outlet_doors												:= TRUE;
	bCloseAllDoors														:= FALSE;
END_IF

IF bExtendAllClamps THEN
	r1.extend_inlet_clamps												:= TRUE;
	r2.extend_inlet_clamps												:= TRUE;
	r3.extend_inlet_clamps												:= TRUE;
	r4.extend_inlet_clamps												:= TRUE;
	r1.extend_outlet_clamps												:= TRUE;
	r2.extend_outlet_clamps												:= TRUE;
	r3.extend_outlet_clamps												:= TRUE;
	r4.extend_outlet_clamps												:= TRUE;
	bExtendAllClamps													:= FALSE;
END_IF

IF bRetractAllClamps THEN
	r1.retract_inlet_clamps												:= TRUE;
	r2.retract_inlet_clamps												:= TRUE;
	r3.retract_inlet_clamps												:= TRUE;
	r4.retract_inlet_clamps												:= TRUE;
	r1.retract_outlet_clamps											:= TRUE;
	r2.retract_outlet_clamps											:= TRUE;
	r3.retract_outlet_clamps											:= TRUE;
	r4.retract_outlet_clamps											:= TRUE;
	bRetractAllClamps													:= FALSE;
END_IF

bAllDoorsOpen															:= r1.doors_open_status AND r2.doors_open_status AND r3.doors_open_status AND r4.doors_open_status;
bAllDoorsClosed															:= r1.doors_closed_status AND r2.doors_closed_status AND r3.doors_closed_status AND r4.doors_closed_status;
bAllClampsExtended														:= r1.clamps_extended_status AND r2.clamps_extended_status AND r3.clamps_extended_status AND r4.clamps_extended_status;
bAllClampsRetracted														:= r1.clamps_retracted_status AND r2.clamps_retracted_status AND r3.clamps_retracted_status AND r4.clamps_retracted_status;

rSorbentHighTemp														:= F_HighestReal(r1.sorbent_high_temp, r2.sorbent_high_temp, r3.sorbent_high_temp, r4.sorbent_high_temp);

bAllDoorsCloseError														:= r1.doors_close_error OR r2.doors_close_error OR r3.doors_close_error OR r4.doors_close_error;
bAllDoorsOpenError														:= r1.doors_open_error OR r2.doors_open_error OR r3.doors_open_error OR r4.doors_open_error;
bAllClampsRetractError													:= r1.clamps_retract_error OR r2.clamps_retract_error OR r3.clamps_retract_error OR r4.clamps_retract_error;
bAllClampsExtendError													:= r1.clamps_extend_error OR r2.clamps_extend_error OR r3.clamps_extend_error OR r4.clamps_extend_error;

// Interlock 7
bILSorbentTempOK														:= rSorbentHighTemp <= SP_maximum_sorbent_temperature OR IL_maximum_sorbent_temperature_or;
rs_error_code_1															:= F_Error(rs_error_code_1, NOT bILSorbentTempOK, errSorbentAboveMaxTemp);
END_ACTION

ACTION A_Process_Adsorption:
// P1 - FB_Reactor_Set.A_Process_Adsorption
// Rev 1.0 - October 29, 2024

CASE current_step OF
	
	0:	;
		
	1:
		rs_adsorption													:= _STARTED;
		M_Step(1);
		
	2:
		M_Step(1);
			
	3:
		M_Step(1);

	4:
		M_Step(1);
			
	5:
		M_Step(1);
		
	6:
		M_Step(1);

	7:
		rTime1															:= 5 * _SECONDS;
		M_Step(1);

	8:
		bTimer1															:= TRUE;
		IF tonTimer1.Q THEN
			M_Step(98);
		END_IF

	96:																														// Reactor error
		rs_error_code_1													:= F_Error(rs_error_code_1, TRUE, errReactor);
		M_Step(1);
		
	97:
		rs_adsorption													:= _ERROR;
		M_Step(99);
		
	98:
		rs_adsorption													:= _COMPLETED;
		M_Step(99);
		
	99:
		A_EAP_Services_Reset();
		M_Step(1);
		
	100:
		bTimer1															:= FALSE;

END_CASE

A_EAP_Services_Check();
END_ACTION

ACTION A_Process_Adsorption_1:
// P1 - FB_Reactor_Set.A_Process_Adsorption_1
// Rev 1.0 - October 29, 2024

CASE current_step OF
	
	0:	;
		
	1:
		rs_adsorption													:= _STARTED;
		M_Step(1);
		
	2:
		steam_control_valve												:= _OPEN;
		steam_control_valve_mode										:= eManual;
		M_Step(1);
			
	3:
		IF steam_control_valve_open THEN
			rTime1														:= 5 * _SECONDS;
			M_Step(1);
		ELSIF steam_control_valve_status = eError THEN
			M_Step(97);
		END_IF

	4:
		bTimer1															:= TRUE;
		IF tonTimer1.Q THEN
			M_Step(1);
		END_IF

	5:
		steam_control_valve												:= _CLOSE;
		steam_control_valve_mode										:= eManual;
		M_Step(1);
		
	6:
		IF steam_control_valve_closed THEN
			rTime1														:= 5 * _SECONDS;
			M_Step(1);
		ELSIF steam_control_valve_status = eError THEN
			M_Step(97);
		END_IF

	7:
		bTimer1															:= TRUE;
		IF tonTimer1.Q THEN
			M_Step(98);
		END_IF

	96:																														// Reactor error
		rs_error_code_1													:= F_Error(rs_error_code_1, TRUE, errReactor);
		M_Step(1);
		
	97:
		rs_adsorption													:= _ERROR;
		M_Step(99);
		
	98:
		rs_adsorption													:= _COMPLETED;
		M_Step(99);
		
	99:
		A_EAP_Services_Reset();
		M_Step(1);
		
	100:
		bTimer1															:= FALSE;

END_CASE

A_EAP_Services_Check();
END_ACTION

ACTION A_Process_Air_Repressurization:
// P1 - FB_Reactor_Set.A_Process_Air_Repressurization
// Rev 1.0 - October 29, 2024

CASE current_step OF
	
	0:	;
		
	1:
		rs_air_repres													:= _STARTED;
		M_Step(1);
		
	2:
		M_Step(1);
			
	3:
		M_Step(1);

	4:
		M_Step(1);
			
	5:
		M_Step(1);
		
	6:
		M_Step(1);

	7:
		rTime1															:= 5 * _SECONDS;
		M_Step(1);

	8:
		bTimer1															:= TRUE;
		IF tonTimer1.Q THEN
			rs_air_repres												:= _COMPLETED;
			M_Step(99);
		END_IF

	96:																														// Reactor error
		rs_error_code_1													:= F_Error(rs_error_code_1, TRUE, errReactor);
		M_Step(99);
		
	97:
		rs_air_repres													:= _ERROR;
		M_Step(99);
		
	98:
		rs_air_repres													:= _COMPLETED;
		M_Step(99);
		
	99:
		A_EAP_Services_Reset();
		M_Step(1);
		
	100:
		bTimer1															:= FALSE;

END_CASE

A_EAP_Services_Check();
END_ACTION

ACTION A_Process_Dead_Air_Evacuation:
// P1 - FB_Reactor_Set.A_Process_Dead_Air_Evacuation
// Rev 1.0 - October 31, 2024

CASE current_step OF
	
	0:	;
		
	1:
		rs_dead_air_evac												:= _STARTED;
		bRetractAllClamps												:= TRUE;
		M_Step(1);
		
	2:
		IF bAllClampsRetracted THEN
			repres_valve												:= FALSE;
			M_Step(1);
		ELSIF bAllClampsRetractError THEN
			M_Step(96);
		END_IF
			
	3:
		IF repres_valve_status = eClear THEN
			bCloseAllDoors												:= TRUE;
			M_Step(1);
		ELSIF repres_valve_status = eError THEN
			M_Step(97);
		END_IF

	4:
		IF bAllDoorsClosed THEN
			bCloseAllValves												:= TRUE;
			M_Step(1);
		ELSIF bAllDoorsCloseError THEN
			M_Step(96);
		END_IF
			
	5:
		IF bAllValvesClear THEN
			rs_dead_air_pump_service_request							:= TRUE;
			M_Step(1);
		ELSIF bValveError THEN
			M_Step(97);
		END_IF
		
	6:
		IF rs_dead_air_pump_service_assigned THEN
			bDeadAirPumpServiceAssigned									:= TRUE;
			IF bILDeadAirValveSorbentTempOk THEN
				dead_air_valve											:= TRUE;
				M_Step(1);
			ELSE
				rs_error_code_1											:= F_Error(rs_error_code_1, TRUE, errDeadAirValveSorbentTempTooHigh);
				M_Step(97);
			END_IF
		END_IF

	7:
		IF dead_air_valve_status = eClear THEN
			rTime1														:= SP_maximum_evacuation_duration * _MINUTES;
			M_Step(1);
		ELSIF dead_air_valve_status = eError THEN
			M_Step(97);
		END_IF

	8:
		bTimer1															:= TRUE;
		IF reactor_pres_error THEN
			M_Step(97);
		ELSIF tonTimer1.Q THEN
			rs_error_code_1												:= F_Error(rs_error_code_1, TRUE, errEvacuationPresFailedToReachTarget);
			M_Step(97);
		ELSIF TIME_TO_REAL(tonTimer1.ET) > (SP_minimum_evacuation_duration * _MINUTES) THEN
			IF reactor_pres < SP_evacuation_target_pressure THEN
				IF SP_evacuation_leak_test_active THEN
					bTimer1												:= FALSE;
					dead_air_valve										:= FALSE;
					A_EAP_Services_Reset();
					rTime1												:= SP_evacuation_leak_test_duration * _MINUTES;
					rEvacLeakTestInitialPressure						:= reactor_pres;
					M_Step(1);
				ELSE
					M_Step(98);
				END_IF
			END_IF
		END_IF

	9:
		bTimer1															:= TRUE;
		IF reactor_pres - rEvacLeakTestInitialPressure > SP_evacuation_leak_test_acceptable_leak THEN
			rs_error_code_1												:= F_Error(rs_error_code_1, TRUE, errReactorLeak);
			M_Step(97);
		ELSIF tonTimer1.Q THEN
			M_Step(98);
		END_IF
		
	96:																														// Reactor error
		rs_error_code_1													:= F_Error(rs_error_code_1, TRUE, errReactor);
		M_Step(1);
		
	97:
		rs_dead_air_evac												:= _ERROR;
		M_Step(99);
		
	98:
		rs_dead_air_evac												:= _COMPLETED;
		M_Step(99);
		
	99:
		dead_air_valve													:= FALSE;
		A_EAP_Services_Reset();
		M_Step(1);
		
	100:
		bTimer1															:= FALSE;

END_CASE

A_EAP_Services_Check();
END_ACTION

ACTION A_Process_Dead_Air_Evacuation_1:
// P1 - FB_Reactor_Set.A_Process_Dead_Air_Evacuation_1
// Rev 1.0 - October 29, 2024

CASE current_step OF
	
	0:	;
		
	1:
		rs_dead_air_evac												:= _STARTED;
		M_Step(1);
		
	2:
		M_Step(1);
			
	3:
		M_Step(1);

	4:
		M_Step(1);
			
	5:
		M_Step(1);
		
	6:
		M_Step(1);

	7:
		rTime1															:= 5 * _SECONDS;
		M_Step(1);

	8:
		bTimer1															:= TRUE;
		IF tonTimer1.Q THEN
			M_Step(99);
		END_IF

	96:																														// Reactor error
		rs_error_code_1													:= F_Error(rs_error_code_1, TRUE, errReactor);
		M_Step(1);
		
	97:
		rs_dead_air_evac												:= _ERROR;
		M_Step(99);
		
	98:
		rs_dead_air_evac												:= _COMPLETED;
		M_Step(99);
		
	99:
		dead_air_valve													:= FALSE;
		A_EAP_Services_Reset();
		M_Step(1);
		
	100:
		bTimer1															:= FALSE;

END_CASE

A_EAP_Services_Check();
END_ACTION

ACTION A_Process_Steam_Desorption:
// P1 - FB_Reactor_Set.A_Process_Steam_Desorption
// Rev 1.0 - October 31, 2024

CASE current_step OF
	
	0:	;
		
	1:
		rs_steam_desorption												:= _STARTED;
		IF reactor_pres > SP_sufficient_desorption_pressure THEN
			rs_error_code_1												:= F_Error(rs_error_code_1, TRUE, errInsufficientDesorptionVacuum);
			M_Step(97);
		ELSE
			bExtendAllClamps											:= TRUE;
			M_Step(1);
		END_IF
		
	2:
		IF bAllClampsExtended THEN
			steam_control_valve_mode									:= eManual;
			steam_control_valve											:= _CLOSE;
			M_Step(1);
		ELSIF bAllClampsExtendError THEN
			M_Step(96);
		END_IF
			
	3:
		IF steam_control_valve_closed THEN
			rs_purge_assist_service_request								:= TRUE;
			rs_vac_cooling_pump_service_request							:= TRUE;
			rs_steam_system_service_request								:= TRUE;
			M_Step(1);
		ELSIF steam_control_valve_status = eError THEN
			M_Step(97);
		END_IF

	4:
		IF rs_purge_assist_service_assigned AND rs_vac_cooling_pump_service_assigned AND rs_steam_system_service_assigned THEN
			bPurgeAssistServiceAssigned									:= TRUE;
			bVacCoolingPumpServiceAssigned								:= TRUE;
			bSteamSystemServiceAssigned									:= TRUE;
			IF bILSteamHeaderValvePresOK THEN
				steam_header_valve										:= TRUE;
				M_Step(1);
			ELSE
			 	rs_error_code_1											:= F_Error(rs_error_code_1, TRUE, errSteamHeaderValvePressureTooHigh);
				M_Step(97);
			END_IF

		END_IF

	5:
		IF steam_header_valve_status = eClear THEN
			rTime1														:= SP_maximum_steam_repressurization_duration * _MINUTES;
			rSteamControlValveSlowMoveIncrement							:= SP_steam_control_valve_slow_move_increment;
			rSteamControlValveSlowMoveFullOpen							:= SP_steam_control_valve_slow_move_full_open;
			steam_control_valve_mode									:= eManual;
			steam_control_valve											:= _OPEN;
			M_Step(1);
		ELSIF steam_header_valve_status = eError THEN
			M_Step(97);
		END_IF
		
	6:
		bTimer1															:= TRUE;
		IF NOT bILReactorPresOK THEN
			M_Step(97);
		ELSIF NOT bILSorbentTempOK THEN
			M_Step(97);
		ELSIF reactor_pres >= SP_steam_repressurization_target_pressure THEN
			bTimer1														:= FALSE;
			purge_valve													:= TRUE;
			M_Step(1);
		ELSIF tontimer1.Q THEN
			IF reactor_pres < SP_acceptable_reactor_pressure THEN
				rs_error_code_1											:= F_Error(rs_error_code_1, TRUE, errInsufficientReactorPressure);
				M_Step(97);
			END_IF
		END_IF
	
	7:
		IF purge_valve_status = eClear THEN
			rTime1														:= SP_purge_duration * _MINUTES;
			steam_control_valve_mode									:= eAuto;
			steam_control_valve_setpoint								:= SP_purge_target_pressure;
			M_Step(1);
		ELSIF purge_valve_status = eError THEN
			M_Step(97);
		END_IF
	
	8:
		bTimer1															:= TRUE;
		rSteamControlValveControlPoint									:= reactor_pres;
		bSteamControlValveControlPointError								:= reactor_pres_error;
		IF NOT bILReactorPresOK THEN
			M_Step(97);
		ELSIF NOT bILSorbentTempOK THEN
			M_Step(97);
		ELSIF tonTimer1.Q THEN
			bTimer1														:= FALSE;
			M_Step(1);
		END_IF
		
	9:
		steam_header_valve												:= FALSE;
		steam_control_valve_mode										:= eManual;
		steam_control_valve												:= _CLOSE;
		purge_valve														:= FALSE;
		M_Step(98);
	
	96:																														// Reactor error
		rs_error_code_1													:= F_Error(rs_error_code_1, TRUE, errReactor);
		M_Step(1);
		
	97:
		rs_steam_desorption												:= _ERROR;
		M_Step(99);
		
	98:
		rs_steam_desorption												:= _COMPLETED;
		M_Step(99);
		
	99:
		A_EAP_Services_Reset();
		M_Step(1);
		
	100:
		bTimer1															:= FALSE;
	
END_CASE

A_EAP_Services_Check();
END_ACTION

ACTION A_Process_Vacuum_Cooling:
// P1 - FB_Reactor_Set.A_Process_Vacuum_Cooling
// Rev 1.0 - October 29, 2024

CASE current_step OF
	
	0:	;
		
	1:
		rs_vacuum_cooling												:= _STARTED;
		rs_vac_cooling_pump_service_request								:= TRUE;
		M_Step(1);
		
	2:
		IF rs_vac_cooling_pump_service_assigned THEN
			bVacCoolingPumpServiceAssigned								:= TRUE;
			cooling_valve												:= TRUE;
			M_Step(1);
		END_IF
			
	3:
		IF cooling_valve_status = eClear THEN
			rTime1														:= SP_maximum_cooling_duration * _MINUTES;
			M_Step(1);
		ELSIF cooling_valve_status = eError THEN
			M_Step(97);
		END_IF

	4:
		bTimer1															:= TRUE;
		IF reactor_pres <= SP_cooling_target_pressure THEN
			M_Step(1);
		ELSIF tonTimer1.Q THEN
			IF reactor_pres <= SP_cooling_acceptable_pressure THEN
				M_Step(1);
			ELSE
				rs_error_code_1											:= F_Error(rs_error_code_1, TRUE, errCoolingPressureTooHigh);
				M_Step(97);
			END_IF
		END_IF
			
	5:
		cooling_valve													:= TRUE;
		bCoolingFailedFirstTry											:= FALSE;
		M_Step(98);
		
	96:																														// Reactor error
		rs_error_code_1													:= F_Error(rs_error_code_1, TRUE, errReactor);
		M_Step(1);
		
	97:
		rs_vacuum_cooling												:= _ERROR;
		M_Step(99);
		
	98:
		rs_vacuum_cooling												:= _COMPLETED;
		M_Step(99);
		
	99:
		A_EAP_Services_Reset();
		M_Step(1);
		
	100:
		bTimer1															:= FALSE;
	
END_CASE

A_EAP_Services_Check();
END_ACTION

ACTION A_Shutdown:
// P1 - FB_Reactor_Set.A_Shutdown
// Rev 1.0 - October 29, 2024

CASE current_step OF
	
	0:	;
		
	1:
		rs_shutdown														:= _STARTED;
		rFanSpeed														:= 0;
		bResetFanSpeed													:= TRUE;
		M_Step(1);
		
	2:
		bCloseAllValves													:= TRUE;
		M_Step(1);
			
	3:
		A_EAP_Services_Reset();
		M_Step(1);

	4:
		bError															:= FALSE;
		IF rSorbentHighTemp > SP_maximum_evac_storage_temperature THEN
			bError														:= TRUE;
			rs_error_code_1												:= F_Error(rs_error_code_1, TRUE, errSorbentAboveMaxStorageTemp);
		END_IF
		IF P_Module.inlet_air_temp > SP_maximum_inlet_air_temperature THEN
			bError														:= TRUE;		
			rs_error_code_1												:= F_Error(rs_error_code_1, TRUE, errInletTempAboveMaxAllowedTemp);
		END_IF
		IF P_Module.inlet_air_temp < SP_minimum_inlet_air_temperature THEN
			bError														:= TRUE;		
			rs_error_code_1												:= F_Error(rs_error_code_1, TRUE, errInletTempBelowMinAllowedTemp);
		END_IF
		rs_shutdown														:= SEL(bError, _COMPLETED, _ERROR);
		M_Step(100);
			
	100:
		bTimer1															:= FALSE;
	
END_CASE
END_ACTION

ACTION A_Shutdown_Estop:
// P1 - FB_Reactor_Set.A_Shutdown_Estop
// Rev 1.0 - October 29, 2024

CASE current_step OF
	
	0:	;
		
	1:
		rs_estop														:= _STARTED;
		M_Step(1);
		
	2:
		M_Step(1);
			
	3:
		M_Step(1);

	4:
		M_Step(1);
			
	5:
		M_Step(1);
		
	6:
		M_Step(1);

	7:
		rTime1															:= 5 * _SECONDS;
		M_Step(1);

	8:
		bTimer1															:= TRUE;
		IF tonTimer1.Q THEN
			rs_estop													:= _COMPLETED;
			M_Step(99);
		END_IF

	97:																														// Reactor error
		rs_error_code_1													:= F_Error(rs_error_code_1, TRUE, errReactor);
		M_Step(1);
		
	98:
		rs_estop														:= _ERROR;
		M_Step(1);
		
	99:
		rs_dead_air_pump_service_request								:= FALSE;
		bDeadAirPumpServiceAssigned											:= FALSE;
		M_Step(1);
		
	100:
		bTimer1															:= FALSE;
	
END_CASE

IF bDeadAirPumpServiceAssigned AND NOT rs_dead_air_pump_service_assigned THEN
	rs_error_code_1														:= F_Error(rs_error_code_1, TRUE, errDeadAirPumpServiceAssignmentLost);
	M_Step(98);
END_IF
END_ACTION

ACTION A_Shutdown_Estop_1:
// P1 - FB_Reactor_Set.A_Shutdown_Estop_1
// Rev 1.0 - October 29, 2024

CASE current_step OF
	
	0:	;
		
	1:
		rs_estop														:= _STARTED;
		M_Step(1);
		
	2:
		M_Step(1);
			
	3:
		M_Step(1);

	4:
		M_Step(1);
			
	5:
		M_Step(1);
		
	6:
		M_Step(1);

	7:
		rTime1															:= 5 * _SECONDS;
		M_Step(1);

	8:
		bTimer1															:= TRUE;
		IF tonTimer1.Q THEN
			rs_estop													:= _COMPLETED;
			M_Step(99);
		END_IF

	97:																														// Reactor error
		rs_error_code_1													:= F_Error(rs_error_code_1, TRUE, errReactor);
		M_Step(1);
		
	98:
		rs_estop														:= _ERROR;
		M_Step(1);
		
	99:
		rs_dead_air_pump_service_request								:= FALSE;
		bDeadAirPumpServiceAssigned											:= FALSE;
		M_Step(1);
		
	100:
		bTimer1															:= FALSE;
	
END_CASE

IF bDeadAirPumpServiceAssigned AND NOT rs_dead_air_pump_service_assigned THEN
	rs_error_code_1														:= F_Error(rs_error_code_1, TRUE, errDeadAirPumpServiceAssignmentLost);
	M_Step(98);
END_IF
END_ACTION

ACTION A_Shutdown_Evac:
// P1 - FB_Reactor_Set.A_Shutdown_Evac
// Rev 1.0 - October 29, 2024

CASE current_step OF
	
	0:	;
		
	1:
		rs_shutdown														:= _STARTED;
		rFanSpeed														:= 0;
		bResetFanSpeed													:= TRUE;
		M_Step(1);
		
	2:
		bCloseAllValves													:= TRUE;
		M_Step(1);
			
	3:
		A_EAP_Services_Reset();
		M_Step(1);

	4:
		bError															:= FALSE;
		IF reactor_pres > SP_maximum_evac_storage_pressure THEN
			bError														:= TRUE;
			rs_error_code_1												:= F_Error(rs_error_code_1, TRUE, errReactorAboveMaxStoragePres);
		END_IF
		rs_shutdown														:= SEL(bError, _COMPLETED, _ERROR);
		M_Step(100);
			
	100:
		bTimer1															:= FALSE;
	
END_CASE
END_ACTION

METHOD M_Step : INT
VAR_INPUT
	Step																: INT;
END_VAR
// P1 - FB_Reactor_Set.M_Step
// Rev 1.0 - October 10, 2024

IF Step = 0 THEN
	current_step														:= 0;
ELSIF Step >= 80 THEN
	current_step														:= Step;
ELSE
	current_step														:= current_step + Step;
END_IF
END_METHOD

METHOD Steam_Desorption_FAT : BOOL
VAR_INPUT
	i_Execute : BOOL;
END_VAR
IF eState  = eSteamDesorption AND i_Execute THEN 
	
	CASE current_step OF
		
		
		1: 
		
			reactor_pres 						:= FAT.st_steam_desorption.step_1.config.react_press;
			SP_sufficient_desorption_pressure 	:= FAT.st_steam_desorption.step_1.config.sp_1;
		
			FAT.st_steam_desorption_result.steps := TO_STRING(current_step);
		
		2: 
		
				
			bAllClampsExtended := bAllClampsExtended OR  STRING_TO_BOOL(FAT.st_steam_desorption.step_2.config.check_1);  
			
			FAT.st_steam_desorption_result.steps := TO_STRING(current_step);
			
		3: 
		
			steam_control_valve_closed := steam_control_valve_closed OR  STRING_TO_BOOL(FAT.st_steam_desorption.step_3.config.valve_1);
			
			FAT.st_steam_desorption_result.steps := TO_STRING(current_step);
				
			
		4 : 
		
			rs_purge_assist_service_assigned 		:= TRUE;
			rs_vac_cooling_pump_service_assigned 	:= TRUE;
			rs_steam_system_service_assigned 		:= TRUE;
			
			reactor_pres 							:= FAT.st_steam_desorption.step_4.config.react_press;
			SP_sufficient_desorption_pressure 		:= FAT.st_steam_desorption.step_4.config.sp_1;
			
			FAT.st_steam_desorption_result.steps := TO_STRING(current_step);
			
		5 :
		
			IF STRING_TO_BOOL(FAT.st_steam_desorption.step_5.config.valve_1) OR steam_header_valve_status = eClear THEN 
				steam_header_valve_status 					:= eClear ;
				SP_maximum_steam_repressurization_duration	:= FAT.st_steam_desorption.step_5.config.sp_1;							
			ELSE
				steam_header_valve_status 					:= eError ;
			END_IF
			
			FAT.st_steam_desorption_result.steps := TO_STRING(current_step);
			
		6 :
		
			
			reactor_pres								:= FAT.st_steam_desorption.step_6.config.react_press;
			SP_maximum_reactor_pressure 				:= FAT.st_steam_desorption.step_6.config.sp_1;
			bILReactorPresOK							:= reactor_pres <= SP_maximum_reactor_pressure;

			rSorbentHighTemp							:= FAT.st_steam_desorption.step_6.config.sorbent_temp;
			SP_maximum_sorbent_temperature				:= FAT.st_steam_desorption.step_6.config.sp_2;
			bILSorbentTempOK							:= rSorbentHighTemp <= SP_maximum_sorbent_temperature;
	
			SP_steam_repressurization_target_pressure 	:= FAT.st_steam_desorption.step_6.config.sp_3;
			
			SP_acceptable_reactor_pressure 				:= FAT.st_steam_desorption.step_6.config.sp_4;
			
			FAT.st_steam_desorption_result.steps := TO_STRING(current_step);
			
		7 : 

			IF STRING_TO_BOOL(FAT.st_steam_desorption.step_7.config.valve_1) OR purge_valve_status = eClear THEN 
				purge_valve_status 	:= eClear ;
				SP_purge_duration 	:= FAT.st_steam_desorption.step_7.config.sp_1;							
			ELSE
				purge_valve_status 	:= eError ;
			END_IF	
			
			FAT.st_steam_desorption_result.steps := TO_STRING(current_step);

		8: 

			reactor_pres								:= FAT.st_steam_desorption.step_8.config.react_press;
			SP_maximum_reactor_pressure 				:= FAT.st_steam_desorption.step_8.config.sp_1;
			bILReactorPresOK							:= reactor_pres <= SP_maximum_reactor_pressure;

			rSorbentHighTemp							:= FAT.st_steam_desorption.step_8.config.sorbent_temp;
			SP_maximum_sorbent_temperature				:= FAT.st_steam_desorption.step_8.config.sp_2;
			bILSorbentTempOK							:= rSorbentHighTemp <= SP_maximum_sorbent_temperature;
			
			FAT.st_steam_desorption_result.steps := TO_STRING(current_step);
					
			
		99 : 
		
			rs_purge_assist_service_assigned := FALSE;
			rs_vac_cooling_pump_service_assigned := FALSE;
			rs_steam_system_service_assigned := FALSE;
			
		100 :
		
			FAT.st_steam_desorption_result.test_name :=  FAT.st_steam_desorption.test_name;
			FAT.st_steam_desorption_result.status := TO_STRING(rs_steam_desorption);
			FAT.st_steam_desorption_result.error := TO_INT(rs_error_code_1);
			current_step := 0;
			
	END_CASE
	
END_IF
END_METHOD

END_FUNCTION_BLOCK

// ---- POUs/FB_Reactor.TcPOU
FUNCTION_BLOCK FB_Reactor
VAR_INPUT
	unit																: INT;
	reset																: BOOL;
	
	{attribute 'OPC.UA.DA' := '1'}  				                
	open_inlet_doors													: BOOL;
	{attribute 'OPC.UA.DA' := '1'}  				                
	close_inlet_doors													: BOOL;
	{attribute 'OPC.UA.DA' := '1'}  				                
	open_outlet_doors													: BOOL;
	{attribute 'OPC.UA.DA' := '1'}  				                
	close_outlet_doors													: BOOL;
	{attribute 'OPC.UA.DA' := '1'}  				                
	extend_inlet_clamps													: BOOL;
	{attribute 'OPC.UA.DA' := '1'}  				                
	retract_inlet_clamps												: BOOL;
	{attribute 'OPC.UA.DA' := '1'}  				                
	extend_outlet_clamps												: BOOL;
	{attribute 'OPC.UA.DA' := '1'}  				                
	retract_outlet_clamps												: BOOL;
	
    /// <summary>VFD01</summary>
	{attribute 'OPC.UA.DA' := '1'}  				                
	fan_vfd																: REAL;
END_VAR
VAR_OUTPUT
	{attribute 'OPC.UA.DA' := '1'}  				                
	{attribute 'OPC.UA.DA.Access' := '1'}  				                
	error_code													AT %Q*	: DWORD;
	{attribute 'OPC.UA.DA' := '1'}  				                
	{attribute 'OPC.UA.DA.Access' := '1'}  				                
	sorbent_low_temp													: REAL;
	{attribute 'OPC.UA.DA' := '1'}  				                
	{attribute 'OPC.UA.DA.Access' := '1'}  				                
	sorbent_high_temp													: REAL;
	{attribute 'OPC.UA.DA' := '1'}  				                
	{attribute 'OPC.UA.DA.Access' := '1'}  				                
	sorbent_average_temp												: REAL;
	{attribute 'OPC.UA.DA' := '1'}  				                
	{attribute 'OPC.UA.DA.Access' := '1'}  				                
	vacuum_cooling_high_temp_count										: INT;
	{attribute 'OPC.UA.DA' := '1'}  				                
	{attribute 'OPC.UA.DA.Access' := '1'}  				                
	adsorption_high_temp_count											: INT;
	{attribute 'OPC.UA.DA' := '1'}  				                
	{attribute 'OPC.UA.DA.Access' := '1'}  				                
	desorption_high_temp_count											: INT;

    /// <summary>TT06</summary>
	{attribute 'OPC.UA.DA' := '1'}  				                
	{attribute 'OPC.UA.DA.Access' := '1'}  				                
	outlet_line_temp													: REAL;						
    /// <summary>TT06</summary>
	{attribute 'OPC.UA.DA' := '1'}  				            	
	{attribute 'OPC.UA.DA.Access' := '1'}  				        	  
	outlet_line_temp_error												: BOOL;

    /// <summary>VFD01</summary>
	{attribute 'OPC.UA.DA' := '1'}  				                
	{attribute 'OPC.UA.DA.Access' := '1'}  				                
	fan_vfd_error														: BOOL;
    /// <summary>VFD01</summary>
	{attribute 'OPC.UA.DA' := '1'}  				                
	{attribute 'OPC.UA.DA.Access' := '1'}  				                
	fan_run_error														: BOOL;
    /// <summary>VFD01</summary>
	{attribute 'OPC.UA.DA' := '1'}  				                
	{attribute 'OPC.UA.DA.Access' := '1'}  				                
	fan_running															: BOOL;

	{attribute 'OPC.UA.DA' := '1'}  				                
	{attribute 'OPC.UA.DA.Access' := '1'}  				                
	inlet_doors_closed_status											: BOOL;
	{attribute 'OPC.UA.DA' := '1'}  				                
	{attribute 'OPC.UA.DA.Access' := '1'}  				                
	inlet_doors_close_error												: BOOL;
	{attribute 'OPC.UA.DA' := '1'}  				                
	inlet_doors_closed_or												: BOOL;
	{attribute 'OPC.UA.DA' := '1'}  				                
	{attribute 'OPC.UA.DA.Access' := '1'}  				                
	inlet_doors_closed_or_status										: BOOL;
	{attribute 'OPC.UA.DA' := '1'}  				                
	{attribute 'OPC.UA.DA.Access' := '1'}  				                
	inlet_doors_open_status												: BOOL;
	{attribute 'OPC.UA.DA' := '1'}  				                
	{attribute 'OPC.UA.DA.Access' := '1'}  				                
	inlet_doors_open_error												: BOOL;
	
	{attribute 'OPC.UA.DA' := '1'}  				                
	{attribute 'OPC.UA.DA.Access' := '1'}  				                
	outlet_doors_closed_status											: BOOL;
	{attribute 'OPC.UA.DA' := '1'}  				                
	{attribute 'OPC.UA.DA.Access' := '1'}  				                
	outlet_doors_close_error											: BOOL;
	{attribute 'OPC.UA.DA' := '1'}  				                
	outlet_doors_closed_or												: BOOL;
	{attribute 'OPC.UA.DA' := '1'}  				                
	{attribute 'OPC.UA.DA.Access' := '1'}  				                
	outlet_doors_closed_or_status										: BOOL;
	{attribute 'OPC.UA.DA' := '1'}  				                
	{attribute 'OPC.UA.DA.Access' := '1'}  				                
	outlet_doors_open_status											: BOOL;
	{attribute 'OPC.UA.DA' := '1'}  				                
	{attribute 'OPC.UA.DA.Access' := '1'}  				                
	outlet_doors_open_error												: BOOL;
	
	doors_closed_status													: BOOL;
	doors_open_status													: BOOL;
	
	doors_open_error													: BOOL;
	doors_close_error													: BOOL;
	
	{attribute 'OPC.UA.DA' := '1'}  				                
	{attribute 'OPC.UA.DA.Access' := '1'}  				                
	inlet_clamps_extended_status										: BOOL;
	{attribute 'OPC.UA.DA' := '1'}  				                
	{attribute 'OPC.UA.DA.Access' := '1'}  				                
	inlet_clamps_extend_error											: BOOL;
	{attribute 'OPC.UA.DA' := '1'}  				                
	{attribute 'OPC.UA.DA.Access' := '1'}  				                
	inlet_clamps_retracted_status										: BOOL;
	{attribute 'OPC.UA.DA' := '1'}  				                
	inlet_clamps_retracted_or											: BOOL;
	{attribute 'OPC.UA.DA' := '1'}  				                
	{attribute 'OPC.UA.DA.Access' := '1'}  				                
	inlet_clamps_retracted_or_status									: BOOL;
	{attribute 'OPC.UA.DA' := '1'}  				                
	{attribute 'OPC.UA.DA.Access' := '1'}  				                
	inlet_clamps_retract_error											: BOOL;

	{attribute 'OPC.UA.DA' := '1'}  				                
	{attribute 'OPC.UA.DA.Access' := '1'}  				                
	outlet_clamps_extended_status										: BOOL;
	{attribute 'OPC.UA.DA' := '1'}  				                
	{attribute 'OPC.UA.DA.Access' := '1'}  				                
	outlet_clamps_extend_error											: BOOL;
	{attribute 'OPC.UA.DA' := '1'}  				                
	{attribute 'OPC.UA.DA.Access' := '1'}  				                
	outlet_clamps_retracted_status										: BOOL;
	{attribute 'OPC.UA.DA' := '1'}  				                
	outlet_clamps_retracted_or											: BOOL;
	{attribute 'OPC.UA.DA' := '1'}  				                
	{attribute 'OPC.UA.DA.Access' := '1'}  				                
	outlet_clamps_retracted_or_status									: BOOL;
	{attribute 'OPC.UA.DA' := '1'}  				                
	{attribute 'OPC.UA.DA.Access' := '1'}  				                
	outlet_clamps_retract_error											: BOOL;

	inlet_clamps_extend_door_open_error									: BOOL;
	outlet_clamps_extend_door_open_error								: BOOL;
	clamps_extend_door_open_error										: BOOL;

	clamps_extended_status												: BOOL;
	clamps_retracted_status												: BOOL;

	clamps_extend_error													: BOOL;
	clamps_retract_error												: BOOL;
END_VAR
VAR
	fbFan																: FB_VFD();
	
	fbInletDoorLeftClosed												: FB_Door_Closed();
	fbInletDoorRightClosed												: FB_Door_Closed();
	fbOutletDoorLeftClosed												: FB_Door_Closed();
	fbOutletDoorRightClosed												: FB_Door_Closed();

	rtrigSorbentErrorCheck												: R_TRIG;
	rtrigExtendInletClamps												: R_TRIG;
	rtrigExtendOutletClamps												: R_TRIG;

